(* CODESYS project CtaSysConfig_2.0.0.0.library
   Description: Config Library der CTA
   Version: 2.0.0.0
   Title: CtaSysConfig
   Author: SIS
   DocFormat: reStructuredText
   Placeholder: CtaSysConfig
   LanguageModelAttribute: qualified-access-only
   DefaultNamespace: CtaSysConfig
   CompiledLibraryCompatibilityVersion: CODESYS V3.5 SP16 Patch 3
   Company: CTA

Project tree, tasks and I/O mapping:
  libraries: VisuDialogs, 3.5.16.20 (System); VisuSymbols, 4.5.0.0 (System); SysTypes2 Interfaces, * (System); Util, 3.5.19.0 (System); Standard, 3.5.18.0 (System); StringUtils, 3.5.20.0 (System); SysFile, 3.5.17.0 (System); SysProcess, 3.5.17.0 (System); SysDir, 3.5.17.0 (System); SysTimeRtc, 3.5.20.0 (System); CtaVisSymbols, 2.0.0.0 (CTA); CtaVisUser, 1.0.0.0 (CTA)
  00000000-0000-0000-0000-000000000000|D:\CoDeSys\LibrariesV3\trunk\Intern\CAA\CAA Template\3.5.2.0 draft\Placeholder.xml
  11 Library Parameter/
  30 Program Organization Units/
    08 Bit/
      function block fbSINT [ST]: proValue, proShowValue, metInit, metNewValue, metNewMinMaxNoSave, metNewValueNoSave, proMin, proMax, proStrPara, metNewMinMax, metCheckState
      function block fbBYTE [ST]: proMin, metNewMinMax, proStrPara, metNewValue, proShowValue, metNewValueNoSave, proMax, proValue, metNewMinMaxNoSave, metInit, metCheckState
      function block fbUSINT [ST]: proMax, metNewValueNoSave, proStrPara, metInit, proShowValue, metNewMinMaxNoSave, proValue, proMin, metNewMinMax, metNewValue, metCheckState
    Basis/
      function block fbBackUpConfig [ST]: actCreateDateTime, actCreateFilePath
      function block fbConfigFile [ST]: metLoad, metOpenFile, proErrorNr, metCodeDirCreate, FB_EXIT, metLoadFile, proEventDetekted, metCheckNr, proFilePathCheckFile, metChild, proLoad, metSaveFile, metSave, proError, proFilePath, metCleanUpInit, metInit, FB_INIT, proSave, proInitDone, ProSetInstancePathOnDynCreate, metCleanUp, metCheckLastChild
      function block fbDataType [ST]: proShowValue, proStateChanged, proIsLoading, metInit, proParaNr, proIsSaving, proSaveOnChange, proStrPara, proChildAddDone, metCheckState
    32 Bit/
      function block fbDWORD [ST]: proMin, proStrPara, metNewMinMax, proShowValue, proValue, metInit, metNewMinMaxNoSave, proMax, metNewValue, metNewValueNoSave, metCheckState
      function block fbREAL [ST]: metNewMinMaxNoSave, metNewValueNoSave, proShowValue, proMin, proStrPara, proMax, metInit, metNewValue, proValue, metNewMinMax, metCheckState
      function block fbUDINT [ST]: metNewMinMaxNoSave, proShowValue, metNewValue, metNewValueNoSave, proValue, metNewMinMax, metInit, proMax, proStrPara, proMin, metCheckState
      function block fbTIME [ST]: proValue, proStrPara, proShowValue, metNewValueNoSave, metNewValue, metInit, metNewMinMax, proMin, metNewMinMaxNoSave, proMax, metCheckState
      function block fbDINT [ST]: proStrPara, metInit, metNewValue, proValue, metNewMinMax, proMin, metNewMinMaxNoSave, proMax, proShowValue, metNewValueNoSave, metCheckState
      function block fbTOD [ST]: proStrPara, metInit, metNewMinMax, proMin, proValue, metNewValueNoSave, metNewMinMaxNoSave, metNewValue, proShowValue, proMax, metCheckState
      function block fbDATE_AND_TIME [ST]: metNewMinMax, proMax, proStrPara, proValue, metInit, proShowValue, metNewMinMaxNoSave, proMin, metNewValue, metNewValueNoSave, metCheckState
    64 Bit/
      function block fbLTIME [ST]: proValue, metNewValue, metInit, proMin, metNewValueNoSave, proShowValue, metNewMinMax, proStrPara, proMax, metNewMinMaxNoSave, metCheckState
    1 Bit/
      function block fbBOOL [ST]: proShowValue, metNewValue, proValue, proStrPara, metInit, metNewValueNoSave, proMax, proMin, metCheckState
    16 Bit/
      function block fbINT [ST]: proShowValue, metNewValueNoSave, metInit, proValue, proMin, proStrPara, proMax, metNewValue, metNewMinMax, metNewMinMaxNoSave, metCheckState
      function block fbWORD [ST]: proMax, proStrPara, metNewValue, proMin, metNewMinMax, metInit, proValue, proShowValue, metNewValueNoSave, metNewMinMaxNoSave, metCheckState
      function block fbUINT [ST]: metNewMinMaxNoSave, proMin, metNewValueNoSave, proMax, proStrPara, proValue, metInit, metNewMinMax, metNewValue, proShowValue, metCheckState
    40 Byte String/
      function block fbSTRING40 [ST]: proStrPara, metNewValueNoSave, metInit, proShowValue, proValue, metNewValue, metCheckState
    Functions/
      function fcFileClose [ST]
      function fcGetMin [ST]
      function fcFileOpen [ST]
      function fcGetValueFromDataType [ST]
      function fcRealToString [ST]
      function fcGetValue [ST]
      function fcGetEnumerationId [ST]
      function fcFillStr [ST]
      function fcGetMax [ST]
      function fcFileDelete [ST]
    function FuGetLocalDateAndTime [ST]
  13 Globale Variablen/
    global variables GVL_Config
  00000000-0000-0000-0000-000000000000|D:\CoDeSys\LibrariesV3\trunk\Intern\CAA\CAA Template\3.4.0.0 draft\Placeholder.xml
  12 Konstanten/
    global variables GlobalKonstant
  40 Visualizations/
    32 Bit/
      UDINT/
        visualisation visUDINT
        visualisation visUDINT_QUERRY
        visualisation visUDINT_ITF
      DINT/
        visualisation visDINT_QUERRY
        visualisation visDINT
        visualisation visDINT_ITF
      REAL/
        visualisation visREAL_QUERRY
        visualisation visREAL
        visualisation visREAL_ITF
      TIME/
        visualisation visTIME
        visualisation visTIME_ITF
        visualisation visTIME_QUERRY
      TOD/
        visualisation visTOD_ITF
        visualisation visTOD
        visualisation visTOD_QUERRY
      DWORD/
        DWORD DEZ/
          visualisation visDWORD_QUERRY_DEZ
          visualisation visDWORD_ITF_DEZ
          visualisation visDWORD_DEZ
        DWORD HEX/
          visualisation visDWORD_HEX
          visualisation visDWORD_ITF_HEX
          visualisation visDWORD_QUERRY_HEX
      DATE AND TIME/
        visualisation visDATE_AND_TIME_ITF
        visualisation visDATE_AND_TIME
        visualisation visDATE_AND_TIME_QUERRY
    8 Bit/
      USINT/
        visualisation visUSINT_QUERRY
        visualisation visUSINT_ITF
        visualisation visUSINT
      BYTE/
        visualisation visBYTE_ITF
        visualisation visBYTE
        visualisation visBYTE_QUERRY
      SINT/
        visualisation visSINT_QUERRY
        visualisation visSINT_ITF
        visualisation visSINT
    16 Bit/
      WORD/
        WORD HEX/
          visualisation visWORD_HEX
          visualisation visWORD_QUERRY_HEX
          visualisation visWORD_ITF_HEX
        WORD DEZ/
          visualisation visWORD_ITF_DEZ
          visualisation visWORD_QUERRY_DEZ
          visualisation visWORD_DEZ
      INT/
        visualisation visINT
        visualisation visINT_ITF
        visualisation visINT_QUERRY
      UINT/
        visualisation visUINT
        visualisation visUINT_ITF
        visualisation visUINT_QUERRY
    40 Byte String/
      visualisation visSTRING40_QUERRY
      visualisation visSTRING40
      visualisation visSTRING40_ITF
    ENUMERATION/
      32 Bit/
        visualisation visENUMERATION_DINT_QUERRY
        visualisation visENUMERATION_DINT
      16 Bit/
        visualisation visENUMERATION_INT
        visualisation visENUMERATION_INT_QUERRY
      visualisation visENUMERATION
      8 Bit/
        visualisation visENUMERATION_BYTE
        visualisation visENUMERATION_BYTE_QUERR
    64 Bit/
      LTIME/
        visualisation visLTIME_ITF
        visualisation visLTIME
        visualisation visLTIME_QUERRY
    1 Bit/
      visualisation visBOOL
      visualisation visBOOL_ITF
      visualisation visBOOL_QUERRY
    Show Data/
      visualisation visSHOWDATA_QUERRY
      visualisation visSHOWDATA
      visualisation visSHOWDATA_ITF
  21 Interface/
    16 Bit/
      interface ITF_WORD: proMax, proMin, proValue
      interface ITF_UINT: proMin, proMax, proValue
      interface ITF_INT: proValue, proMin, proMax
    1 Bit/
      interface ITF_BOOL: proValue
    32 Bit/
      interface ITF_REAL: proValue, proMax, proMin
      interface ITF_TIME: proValue, proMax, proMin
      interface ITF_TOD: proValue, proMin, proMax
      interface ITF_DATE_AND_TIME: proMax, proValue, proMin
      interface ITF_UDINT: proMin, proMax, proValue
      interface ITF_DINT: proMax, proMin, proValue
      interface ITF_DWORD: proMin, proValue, proMax
    08 Bit/
      interface ITF_SINT: proValue, proMax, proMin
      interface ITF_BYTE: proMax, proValue, proMin
      interface ITF_USINT: proMin, proValue, proMax
    40 Byte String/
      interface ITF_STRING40: proValue
    Basis/
      interface ITF_DATATYPE: proStrPara, proChildAddDone, proStateChanged, proShowValue, proIsSaving, metInit, proSaveOnChange, proParaNr, proIsLoading
      interface ITF_CONFIGFILE: proLoad, metInit, metSave, proInitDone, metLoad, proSave, metCheckLastChild
    64 Bit/
      interface ITF_LTIME: proValue, proMin, proMax
  60 Textlisten/
  20 Structs/
    data type scStateDataType
    data type scStateConfigFile
  text list GlobalTextList
  50 Images/
  10 Documenation/
    global variables VersionHistory
    global variables readMe
  00000000-0000-0000-0000-000000000000|D:\CoDeSys\LibrariesV3\trunk\Intern\CAA\CAA Template\3.2.0.3 draft\Prefix.pdf
*)

// 20 Structs/scStateDataType
TYPE scStateDataType :
    STRUCT
        xInitDoneDataType       :   BIT;
        xInitDoneConfig         :   BIT;
        xUpdateOldValueNoSave   :   BIT;
        xSaveOnChange           :   BIT; 
        xIsSaving               :   BIT;
        xIsLoading              :   BIT; 
		xStateChanged			:	BIT;  
		xChildAddDone			:	BIT;
    END_STRUCT
END_TYPE

// 20 Structs/scStateConfigFile
TYPE scStateConfigFile :
    STRUCT
        xInit                   :   BIT;
		xInitDone				:	BIT;
		xGetChild				:	BIT;
        xEventSave              :   BIT;
        xEventLoad              :   BIT;
        xEventDetekted          :   BIT;
        xIsOpen                 :   BIT;        
    END_STRUCT
END_TYPE

// 12 Konstanten/GlobalKonstant
{attribute 'qualified_only'}
VAR_GLOBAL CONSTANT
    usiFeldLeng     :   USINT   :=    40;
    diStringSize    :   UINT    :=   129;
    diLineSize      :   UINT    :=   131;    
END_VAR

// 10 Documenation/VersionHistory
(* 

.. image:: ../../Images/CTA_Logo.jpg
   :align: right
   :width: 15% 

**Vorlage**   


============ =========== =========== ============================================
**Date**     **Version** **Author**  **Change**
------------ ----------- ----------- --------------------------------------------
04.03.2021   0.0.0.0     SIS         Vorlage erstellt

============ =========== =========== ============================================


*)
VAR_GLOBAL
    stInfo : STRING:= '0.0.0.0, Vorlage, CTA';
END_VAR

// 10 Documenation/readMe
(*

**ReadMe**
 
|	**Empfehlung**
|
|	Dokumentrieren Sie die Library für eine nachhaltige Entwicklung
|     
| *Beispiel*
| 
| Dies ist die Vorlage Library der CTA. Erstellen Sie ihre Library anhand dieser Vorlage.
*)

VAR_GLOBAL
    xReadMeDone              :   BOOL;
END_VAR

// 13 Globale Variablen/GVL_Config
{attribute 'qualified_only'}
VAR_GLOBAL
    stBackUp            :   STRING[30];
    xSave               :   BOOL;
    xLoad               :   BOOL;
    xError              :   BOOL;
    stPath              :   STRING[255];
END_VAR

// 30 Program Organization Units/32 Bit/fbDWORD
FUNCTION_BLOCK fbDWORD EXTENDS fbDataType IMPLEMENTS ITF_DWORD
VAR_INPUT CONSTANT
    _WertInit      :   DWORD;
    _MinInit       :   DWORD;
    _MaxInit       :   DWORD;       
END_VAR
VAR
    dwValue          :   DWORD;   
    dwMin            :   DWORD;
    dwMax            :   DWORD; 
    {attribute 'hide'}
    dwValueOld       :   DWORD; 
    {attribute 'hide'}
    dwMinOld         :   DWORD;
    {attribute 'hide'}
    dwMaxOld         :   DWORD;
END_VAR

(* Call Supper Objekt *)
IF itfConfigFb <> 0 THEN
    SUPER^();
END_IF;

{attribute 'monitoring':='call'}
PROPERTY proMin : DWORD
SET
dwMin := LIMIT(16#0,proMin,16#FFFFFFFF);
END_SET
GET
proMin := dwMin;
END_GET
END_PROPERTY

{attribute 'hide'}
{attribute 'monitoring':='call'}
PROPERTY proStrPara : STRING(129)
// {attribute 'hide'}
SET
proMax    := TO_DWORD(fcGetMax  ( proStrPara));
proMin    := TO_DWORD(fcGetMin  ( proStrPara));
proValue  := TO_DWORD(fcGetValue( proStrPara));
END_SET
GET
proStrPara :=   CONCAT(                    
                CONCAT( 
                CONCAT(
                CONCAT(                 
                CONCAT(                    
                CONCAT( fcfillStr(CONCAT('P',TO_STRING(SUPER^._usiParaNr)),6)       ,
                        ';'                                                         ),
                        fcfillStr(TO_STRING(dwValue),GlobalKonstant.usiFeldLeng)    ),
                        ';'                                                         ),
                        fcfillStr(TO_STRING(dwMin),GlobalKonstant.usiFeldLeng)      ),
                        ';'                                                         ),
                        fcfillStr(TO_STRING(dwMax),GlobalKonstant.usiFeldLeng)      );
END_GET
END_PROPERTY

METHOD metNewMinMax : BOOL
VAR_INPUT
    newMin      :   DWORD;
    newMax      :   DWORD;
END_VAR
IF newMin <> newMax THEN
    proMin      := newMin;
    proMax      := newMax;
    proValue    := dwValue;    
END_IF;
metNewMinMax := TRUE;
END_METHOD

PROPERTY proShowValue : STRING[40]
GET
proShowValue := TO_STRING(dwValue);
END_GET
END_PROPERTY

{attribute 'monitoring':='call'}
PROPERTY proValue : DWORD
GET
proValue := dwValue;
END_GET
SET
dwValue := LIMIT(proMin,proValue,proMax);
END_SET
END_PROPERTY

{attribute 'hide'}
METHOD metInit : BOOL
IF _MinInit <> _MaxInit THEN
    proMin    := _MinInit;
    proMax    := _MaxInit;
ELSE
    proMin    := 16#F;
    proMax    := 16#FFFFFFFF;
END_IF;
    proValue  := _WertInit;
END_METHOD

METHOD metNewMinMaxNoSave : BOOL
VAR_INPUT
    newMinNoSave      :   DWORD;
    newMaxNoSave      :   DWORD;
END_VAR
IF newMinNoSave <> newMaxNoSave THEN
    proMin      := newMinNoSave;
    proMax      := newMaxNoSave;
    proValue    := dwValue;    
    scState.xUpdateOldValueNoSave := TRUE;
END_IF;
metNewMinMaxNoSave := TRUE;
END_METHOD

{attribute 'monitoring':='call'}
PROPERTY proMax : DWORD
SET
dwMax := LIMIT(16#0,proMax,16#FFFFFFFF);
END_SET
GET
proMax := dwMax;
END_GET
END_PROPERTY

METHOD metNewValue : BOOL
VAR_INPUT
    newValue   :   DWORD;
END_VAR
proValue := newValue;
metNewValue := TRUE;
END_METHOD

METHOD metNewValueNoSave : BOOL
VAR_INPUT
    newValueNoSave   :   DWORD;
END_VAR
proValue := newValueNoSave;
scState.xUpdateOldValueNoSave := TRUE;
metNewValueNoSave := TRUE;
END_METHOD

{attribute 'hide'}
METHOD metCheckState : BOOL
(* Search Change & Save Old Values *)
IF dwValue <> dwValueOld OR dwMin <> dwMinOld OR dwMax <> dwMaxOld OR scState.xUpdateOldValueNoSave THEN
    (* Prüfen ob die Werte bei änderung gespeichert werden sollen *)
    IF scState.xUpdateOldValueNoSave THEN
        scState.xUpdateOldValueNoSave := FALSE;
    ELSE
        proSaveOnChange 	:= TRUE;
	END_IF
	(*State Changed*) 
	scState.xStateChanged 	:= TRUE;   
    proValue   				:= dwValue;
    dwValueOld 				:= proValue;
    proMin     				:= dwMin;
    proMax     				:= dwMax;        
    dwMinOld   				:= proMin;
    dwMaxOld   				:= proMax;
ELSE
	(*State Changed*) 
	scState.xStateChanged 	:= FALSE;    
END_IF;
END_METHOD

END_FUNCTION_BLOCK

// 30 Program Organization Units/Basis/fbDataType
{attribute 'hide_all_locals'}
FUNCTION_BLOCK fbDataType IMPLEMENTS ITF_DATATYPE
VAR_INPUT
    _usiParaNr              :   USINT;
    itfConfigFb             :   ITF_CONFIGFILE;   
END_VAR
VAR
    scState                 :   scStateDataType;
    itfConfigFbSync         :   ITF_CONFIGFILE;
END_VAR

IF itfConfigFb <> 0 THEN
	IF itfConfigFbSync = 0 THEN
		__QUERYINTERFACE(itfConfigFb,itfConfigFbSync);
	END_IF;
	IF itfConfigFb = itfConfigFbSync THEN
		THIS^.metCheckState();
		IF NOT scState.xInitDoneDataType THEN
			THIS^.metInit();
			scState.xInitDoneDataType := TRUE;
		END_IF;
		IF itfConfigFb.proInitDone THEN    
			IF itfConfigFb.proLoad THEN
				itfConfigFb.metLoad(THIS^);
			END_IF;
			IF itfConfigFb.proSave OR scState.xSaveOnChange THEN
				itfConfigFb.metSave(THIS^);
			END_IF;
			itfConfigFb.metCheckLastChild(THIS^);
		ELSIF NOT scState.xInitDoneConfig THEN
			IF itfConfigFb.metInit(THIS^) THEN
				scState.xInitDoneConfig         := TRUE;
				scState.xUpdateOldValueNoSave   := TRUE;
			END_IF;
		END_IF;
	END_IF;    
END_IF;
(* Delete itfConfigFb *)
itfConfigFb := 0;

PROPERTY proShowValue : STRING[40]
GET
proShowValue := '';
END_GET
END_PROPERTY

{attribute 'monitoring':='call'}
PROPERTY proStateChanged : BOOL
GET
proStateChanged := scState.xStateChanged;
END_GET
END_PROPERTY

PROPERTY proIsLoading : BOOL
SET
scState.xIsLoading :=proIsLoading;
END_SET
GET
proIsLoading := scState.xIsLoading;
END_GET
END_PROPERTY

{attribute 'hide'}
METHOD metInit : BOOL
END_METHOD

{attribute 'monitoring':='call'}
PROPERTY proParaNr : USINT
GET
proParaNr := LIMIT(1,_usiParaNr,255);
END_GET
END_PROPERTY

PROPERTY proIsSaving : BOOL
SET
scState.xIsSaving := proIsSaving;
END_SET
GET
proIsSaving := scState.xIsSaving;
END_GET
END_PROPERTY

{attribute 'hide'}
{attribute 'monitoring':='call'}
PROPERTY proSaveOnChange : BOOL
SET
scState.xSaveOnChange := proSaveOnChange;
END_SET
GET
proSaveOnChange := scState.xSaveOnChange;
END_GET
END_PROPERTY

{attribute 'hide'}
{attribute 'monitoring':='call'}
PROPERTY proStrPara : STRING[129]
SET
END_SET
GET
END_GET
END_PROPERTY

PROPERTY proChildAddDone : BOOL
SET
scState.xChildAddDone := proChildAddDone;
END_SET
GET
proChildAddDone := scState.xChildAddDone;
END_GET
END_PROPERTY

{attribute 'hide'}
METHOD metCheckState : BOOL
END_METHOD

END_FUNCTION_BLOCK

// 21 Interface/Basis/ITF_DATATYPE
INTERFACE ITF_DATATYPE EXTENDS __SYSTEM.IQueryInterface

{attribute 'hide'}
{attribute 'monitoring':='call'}
PROPERTY proStrPara : STRING[129]
// {attribute 'hide'}
(*
(* Get *)
(* Tabellenaufbau
+-----+------+------+------+
| PNr | Wert | Min  | Max  |
+-----+------+------+------+
| 6By ; 40By ; 40By ; 40By | = 129By
+-----+------+------+------+
*)
proStrPara :=   CONCAT(                    
                CONCAT( 
                CONCAT(
                CONCAT(                 
                CONCAT(                    
                CONCAT( fcfillStr(CONCAT('P',TO_STRING(_usiParaNr)),5)  ,
                        ';'                                                 ),
                        fcfillStr(TO_STRING(rValue),Konstant.usiFeldLeng)   ),
                        ';'                                                 ),
                        fcfillStr(TO_STRING(rMin),Konstant.usiFeldLeng)     ),
                        ';'                                                 ),
                        fcfillStr(TO_STRING(rMax),Konstant.usiFeldLeng)     );    
                        
                        
                        
(* Set *)
rValue  := TO_REAL(MID(proStrPara,Konstant.usiFeldLeng,7 + (Konstant.usiFeldLeng * 1)+ 0));
rMin    := TO_REAL(MID(proStrPara,Konstant.usiFeldLeng,7 + (Konstant.usiFeldLeng * 2)+ 1));
rMax    := TO_REAL(MID(proStrPara,Konstant.usiFeldLeng,7 + (Konstant.usiFeldLeng * 3)+ 2));                      
                                                
*)
SET
END_SET
GET
END_GET
END_PROPERTY

PROPERTY proChildAddDone : BOOL
GET
END_GET
SET
END_SET
END_PROPERTY

{attribute 'monitoring':='call'}
PROPERTY proStateChanged : BOOL
GET
END_GET
END_PROPERTY

PROPERTY proShowValue : STRING[40]
GET
END_GET
END_PROPERTY

PROPERTY proIsSaving : BOOL
GET
END_GET
SET
END_SET
END_PROPERTY

{attribute 'hide'}
METHOD metInit : BOOL
VAR_INPUT
END_VAR
END_METHOD

{attribute 'monitoring':='call'}
PROPERTY proSaveOnChange : BOOL
SET
END_SET
GET
END_GET
END_PROPERTY

{attribute 'hide'}
{attribute 'monitoring':='call'}
PROPERTY proParaNr : USINT
GET
END_GET
END_PROPERTY

PROPERTY proIsLoading : BOOL
GET
END_GET
SET
END_SET
END_PROPERTY

END_INTERFACE

// 30 Program Organization Units/Functions/fcFillStr
FUNCTION fcFillStr : STRING[GlobalKonstant.usiFeldLeng]
VAR_INPUT
	{attribute 'monitoring_encoding' := 'UTF-8'}
    stIn           : STRING[GlobalKonstant.usiFeldLeng];
    uiLen          : UINT;
END_VAR
VAR
    ui : UINT;
END_VAR

fcFillStr := '';
fcFillStr := stIn;
IF TO_UINT(LEN(stIn)) < uiLen THEN
    FOR ui := LIMIT(0,TO_UINT(LEN(stIn)),LIMIT(0,uiLen,GlobalKonstant.usiFeldLeng)) TO LIMIT(0,uiLen-1,GlobalKonstant.usiFeldLeng) DO
        IF ui = TO_UINT(LEN(stIn)) THEN
            fcFillStr[ui]       := 124; // Trennzeichen
        ELSE
            fcFillStr[ui]       := 32;  // Lehrzeichen
        END_IF; 
        fcFillStr[ui+1]     := 0;  // ClearByte
    END_FOR;
END_IF;

END_FUNCTION

// 21 Interface/Basis/ITF_CONFIGFILE
INTERFACE ITF_CONFIGFILE EXTENDS __SYSTEM.IQueryInterface

{attribute 'monitoring':='call'}
PROPERTY proLoad : BOOL
GET
END_GET
END_PROPERTY

METHOD metInit : BOOL
VAR_INPUT
    itfDataTypeObj  :   ITF_DATATYPE;
END_VAR
END_METHOD

METHOD metSave : BOOL
VAR_INPUT
    itfDataTypeObj  :   ITF_DATATYPE;
END_VAR
END_METHOD

{attribute 'monitoring':='call'}
PROPERTY proInitDone : BOOL
GET
END_GET
END_PROPERTY

METHOD metLoad : BOOL
VAR_INPUT
    itfDataTypeObj  :   ITF_DATATYPE;
END_VAR
END_METHOD

{attribute 'monitoring':='call'}
PROPERTY proSave : BOOL
GET
END_GET
END_PROPERTY

METHOD metCheckLastChild
VAR_INPUT  
    itfDataTypeObj  :   ITF_DATATYPE;
END_VAR
END_METHOD

END_INTERFACE

// 21 Interface/32 Bit/ITF_DWORD
INTERFACE ITF_DWORD EXTENDS ITF_DATATYPE

{attribute 'monitoring':='call'}
PROPERTY proMin : DWORD
SET
END_SET
GET
END_GET
END_PROPERTY

{attribute 'monitoring':='call'}
PROPERTY proValue : DWORD
SET
END_SET
GET
END_GET
END_PROPERTY

{attribute 'monitoring':='call'}
PROPERTY proMax : DWORD
GET
END_GET
SET
END_SET
END_PROPERTY

END_INTERFACE

// 30 Program Organization Units/Functions/fcGetMax
FUNCTION fcGetMax : STRING[40]
VAR_INPUT
	{attribute 'monitoring_encoding' := 'UTF-8'}
    stStrPara   :   STRING[170];    
END_VAR
VAR
END_VAR

fcGetMax                    := (MID(stStrPara,GlobalKonstant.usiFeldLeng,7 + (GlobalKonstant.usiFeldLeng * 2)+ 3));
(* Abschlusszeichen Finden *)
IF FIND(fcGetMax,'|') <> 0 THEN
    fcGetMax                := LEFT(fcGetMax,FIND(fcGetMax,'|')-1);
END_IF;
fcGetMax[LEN(fcGetMax)]     := 0;

END_FUNCTION

// 30 Program Organization Units/Functions/fcGetMin
FUNCTION fcGetMin : STRING[40]
VAR_INPUT
	{attribute 'monitoring_encoding' := 'UTF-8'}
    stStrPara   :   STRING[170];    
END_VAR
VAR
END_VAR

fcGetMin                    := (MID(stStrPara,GlobalKonstant.usiFeldLeng,7 + (GlobalKonstant.usiFeldLeng * 1)+ 2));
(* Abschlusszeichen Finden *)
IF FIND(fcGetMin,'|') <> 0 THEN
    fcGetMin                := LEFT(fcGetMin,FIND(fcGetMin,'|')-1);
END_IF;
fcGetMin[LEN(fcGetMin)]     := 0;

END_FUNCTION

// 30 Program Organization Units/Functions/fcGetValue
{attribute 'hide'}
FUNCTION fcGetValue : STRING[GlobalKonstant.usiFeldLeng]
VAR_INPUT
	{attribute 'monitoring_encoding' := 'UTF-8'}
    stStrPara   :   STRING[126];
END_VAR
VAR
END_VAR

fcGetValue                      := MID(stStrPara,GlobalKonstant.usiFeldLeng,7 + 1);
(* Abschlusszeichen Finden *)
IF FIND(fcGetValue,'|') <> 0 THEN
    fcGetValue                  := LEFT(fcGetValue,FIND(fcGetValue,'|')-1);   
END_IF;
fcGetValue[LEN(fcGetValue)]     := 0;

END_FUNCTION

// 30 Program Organization Units/08 Bit/fbSINT
FUNCTION_BLOCK fbSINT EXTENDS fbDataType IMPLEMENTS ITF_SINT
VAR_INPUT CONSTANT
    _WertInit      :   SINT;
    _MinInit       :   SINT;
    _MaxInit       :   SINT;       
END_VAR
VAR
    siValue          :   SINT;   
    siMin            :   SINT;
    siMax            :   SINT; 
    {attribute 'hide'}
    siValueOld       :   SINT;
    {attribute 'hide'}
    siMinOld         :   SINT;
    {attribute 'hide'}
    siMaxOld         :   SINT; 
END_VAR

(* Call Supper Objekt *)
IF itfConfigFb <> 0 THEN
    SUPER^();
END_IF;

{attribute 'monitoring':='call'}
PROPERTY proValue : sINT
SET
siValue := LIMIT(proMin,proValue,proMax);
END_SET
GET
proValue := siValue;
END_GET
END_PROPERTY

PROPERTY proShowValue : STRING[40]
GET
proShowValue := TO_STRING(siValue);
END_GET
END_PROPERTY

{attribute 'hide'}
METHOD metInit : BOOL
IF _MinInit <> _MaxInit THEN
    proMin    := _MinInit;
    proMax    := _MaxInit;
ELSE
    proMin    :=  -128;
    proMax    :=   127;
END_IF;
    proValue  := _WertInit;
END_METHOD

METHOD metNewValue : BOOL
VAR_INPUT
    newValue   :   SINT;
END_VAR
proValue := newValue;
metNewValue := TRUE;
END_METHOD

METHOD metNewMinMaxNoSave : BOOL
VAR_INPUT
    newMinNoSave      :   SINT;
    newMaxNoSave      :   SINT;
END_VAR
IF newMinNoSave <> newMaxNoSave THEN
    proMin      := newMinNoSave;
    proMax      := newMaxNoSave;
    proValue    := siValue;    
    scState.xUpdateOldValueNoSave := TRUE;
END_IF;
metNewMinMaxNoSave := TRUE;
END_METHOD

METHOD metNewValueNoSave : BOOL
VAR_INPUT
    newValueNoSave   :   SINT;
END_VAR
proValue := newValueNoSave;
scState.xUpdateOldValueNoSave := TRUE;
metNewValueNoSave := TRUE;
END_METHOD

{attribute 'monitoring':='call'}
PROPERTY proMin : sINT
SET
siMin := LIMIT(-128,proMin,127);
END_SET
GET
proMin := siMin;
END_GET
END_PROPERTY

{attribute 'monitoring':='call'}
PROPERTY proMax : sINT
GET
proMax := siMax;
END_GET
SET
siMax := LIMIT(-128,proMax,127);
END_SET
END_PROPERTY

{attribute 'hide'}
{attribute 'monitoring':='call'}
PROPERTY proStrPara : STRING(129)
// {attribute 'hide'}
SET
proMax    := TO_SINT(fcGetMax  ( proStrPara));
proMin    := TO_SINT(fcGetMin  ( proStrPara));
proValue  := TO_SINT(fcGetValue( proStrPara));
END_SET
GET
proStrPara :=   CONCAT(                    
                CONCAT( 
                CONCAT(
                CONCAT(                 
                CONCAT(                    
                CONCAT( fcfillStr(CONCAT('P',TO_STRING(SUPER^._usiParaNr)),6)    ,
                        ';'                                                     ),
                        fcfillStr(TO_STRING(siValue),GlobalKonstant.usiFeldLeng)),
                        ';'                                                     ),
                        fcfillStr(TO_STRING(siMin),GlobalKonstant.usiFeldLeng)  ),
                        ';'                                                     ),
                        fcfillStr(TO_STRING(siMax),GlobalKonstant.usiFeldLeng)  );
END_GET
END_PROPERTY

METHOD metNewMinMax : BOOL
VAR_INPUT
    newMin      :   SINT;
    newMax      :   SINT;
END_VAR
IF newMin <> newMax THEN
    proMin      := newMin;
    proMax      := newMax;
    proValue    := siValue;    
END_IF;
metNewMinMax := TRUE;
END_METHOD

{attribute 'hide'}
METHOD metCheckState : BOOL
(* Search Change & Save Old Values *)
IF siValue <> siValueOld OR siMin <> siMinOld OR siMax <> siMaxOld OR scState.xUpdateOldValueNoSave THEN
    (* Prüfen ob die Werte bei änderung gespeichert werden sollen *)
    IF scState.xUpdateOldValueNoSave THEN
        scState.xUpdateOldValueNoSave := FALSE;
    ELSE
        proSaveOnChange 	:= TRUE;
	END_IF
	(*State Changed*) 
	scState.xStateChanged 	:= TRUE;   
    proValue  				:= siValue;
    siValueOld 				:= proValue;
    proMin     				:= siMin;
    proMax     				:= siMax;    
    siMinOld   				:= proMin;
    siMaxOld   				:= proMax;
ELSE
	(*State Changed*) 
	scState.xStateChanged 	:= FALSE;    
END_IF;
END_METHOD

END_FUNCTION_BLOCK

// 21 Interface/08 Bit/ITF_SINT
INTERFACE ITF_SINT EXTENDS ITF_DATATYPE

{attribute 'monitoring':='call'}
PROPERTY proValue : sINT
SET
END_SET
GET
END_GET
END_PROPERTY

{attribute 'monitoring':='call'}
PROPERTY proMax : sINT
SET
END_SET
GET
END_GET
END_PROPERTY

{attribute 'monitoring':='call'}
PROPERTY proMin : sINT
GET
END_GET
SET
END_SET
END_PROPERTY

END_INTERFACE

// 30 Program Organization Units/32 Bit/fbREAL
FUNCTION_BLOCK fbREAL EXTENDS fbDataType IMPLEMENTS ITF_REAL
VAR_INPUT CONSTANT
    _WertInit      :   REAL;
    _MinInit       :   REAL;
    _MaxInit       :   REAL;       
END_VAR
VAR
    rValue          :   REAL;   
    rMin            :   REAL;
    rMax            :   REAL; 
    {attribute 'hide'}
    rValueOld       :   REAL; 
    {attribute 'hide'}
    rMinOld         :   REAL;
    {attribute 'hide'}
    rMaxOld         :   REAL;
END_VAR

(* Call Supper Objekt *)
IF itfConfigFb <> 0 THEN
    SUPER^();
END_IF;

METHOD metNewMinMaxNoSave : BOOL
VAR_INPUT
    newMinNoSave      :   REAL;
    newMaxNoSave      :   REAL;
END_VAR
IF newMinNoSave <> newMaxNoSave THEN
    proMin      := newMinNoSave;
    proMax      := newMaxNoSave;
    proValue    := rValue;    
    scState.xUpdateOldValueNoSave := TRUE;
END_IF;
metNewMinMaxNoSave := TRUE;
END_METHOD

METHOD metNewValueNoSave : BOOL
VAR_INPUT
    newValueNoSave   :   REAL;
END_VAR
proValue := newValueNoSave;
scState.xUpdateOldValueNoSave := TRUE;
metNewValueNoSave := TRUE;
END_METHOD

PROPERTY proShowValue : STRING[40]
GET
proShowValue := TO_STRING(rValue);
END_GET
END_PROPERTY

{attribute 'monitoring':='call'}
PROPERTY proMin : REAL
SET
rMin := LIMIT(-3.402823E+38,proMin,3.402823E+38);
END_SET
GET
proMin := rMin;
END_GET
END_PROPERTY

{attribute 'hide'}
{attribute 'monitoring':='call'}
PROPERTY proStrPara : STRING[129]
GET
proStrPara :=   CONCAT(                    
                CONCAT( 
                CONCAT(
                CONCAT(                 
                CONCAT(                    
                CONCAT( fcfillStr(CONCAT('P',TO_STRING(SUPER^._usiParaNr)),6)       ,
                        ';'                                                         ),
                        fcfillStr(TO_STRING(rValue),GlobalKonstant.usiFeldLeng)     ),
                        ';'                                                         ),
                        fcfillStr(TO_STRING(rMin),GlobalKonstant.usiFeldLeng)       ),
                        ';'                                                         ),
                        fcfillStr(TO_STRING(rMax),GlobalKonstant.usiFeldLeng)       );
END_GET
SET
proMax    := TO_REAL(fcGetMax  ( proStrPara));
proMin    := TO_REAL(fcGetMin  ( proStrPara));
proValue  := TO_REAL(fcGetValue( proStrPara));
END_SET
END_PROPERTY

{attribute 'monitoring':='call'}
PROPERTY proMax : REAL
SET
rMax := LIMIT(-3.402823E+38,proMax,3.402823E+38);
END_SET
GET
proMax := rMax;
END_GET
END_PROPERTY

{attribute 'hide'}
METHOD metInit : BOOL
IF _MinInit <> _MaxInit THEN
    proMin    := _MinInit;
    proMax    := _MaxInit;
ELSE
    proMin    := -3.402823E+38;
    proMax    :=  3.402823E+38;
END_IF;
    proValue  := _WertInit;
END_METHOD

METHOD metNewValue : BOOL
VAR_INPUT
    newValue   :   REAL;
END_VAR
proValue := newValue;
metNewValue := TRUE;
END_METHOD

{attribute 'monitoring':='call'}
PROPERTY proValue : REAL
SET
rValue := LIMIT(proMin,proValue,proMax);
END_SET
GET
proValue := LIMIT(rMin,rValue,rMax);
END_GET
END_PROPERTY

METHOD metNewMinMax : BOOL
VAR_INPUT
    newMin      :   REAL;
    newMax      :   REAL;
END_VAR
IF newMin <> newMax THEN
    proMin      := newMin;
    proMax      := newMax;
    proValue    := rValue;    
END_IF;
metNewMinMax := TRUE;
END_METHOD

{attribute 'hide'}
METHOD metCheckState : BOOL
(* Search Change & Save Old Values *)
IF rValue <> rValueOld OR rMin <> rMinOld OR rMax <> rMaxOld OR scState.xUpdateOldValueNoSave THEN
    (* Prüfen ob die Werte bei änderung gespeichert werden sollen *)
    IF scState.xUpdateOldValueNoSave THEN
        scState.xUpdateOldValueNoSave := FALSE;
    ELSE
        proSaveOnChange 	:= TRUE;
	END_IF
	(*State Changed*) 
	scState.xStateChanged 	:= TRUE;   
    proValue  				:= rValue;
    rValueOld 				:= proValue;
    proMin    				:= rMin;
    proMax    				:= rMax;      
    rMinOld   				:= proMin;
    rMaxOld   				:= proMax;
ELSE
	(*State Changed*) 
	scState.xStateChanged 	:= FALSE;      
END_IF;
END_METHOD

END_FUNCTION_BLOCK

// 21 Interface/32 Bit/ITF_REAL
INTERFACE ITF_REAL EXTENDS ITF_DATATYPE

{attribute 'monitoring':='call'}
PROPERTY proValue : REAL
SET
END_SET
GET
END_GET
END_PROPERTY

{attribute 'monitoring':='call'}
PROPERTY proMax : REAL
SET
END_SET
GET
END_GET
END_PROPERTY

{attribute 'monitoring':='call'}
PROPERTY proMin : REAL
SET
END_SET
GET
END_GET
END_PROPERTY

END_INTERFACE

// 30 Program Organization Units/08 Bit/fbBYTE
FUNCTION_BLOCK fbBYTE EXTENDS fbDataType IMPLEMENTS ITF_BYTE
VAR_INPUT CONSTANT
    _WertInit        :   BYTE;
    _MinInit         :   BYTE;
    _MaxInit         :   BYTE;       
END_VAR
VAR
    byValue          :   BYTE;   
    byMin            :   BYTE;
    byMax            :   BYTE; 
    {attribute 'hide'} 
    byValueOld       :   BYTE; 
    {attribute 'hide'} 
    byMinOld         :   BYTE;
    {attribute 'hide'} 
    byMaxOld         :   BYTE; 
END_VAR

(* Call Supper Objekt *)
IF itfConfigFb <> 0 THEN
    SUPER^();
END_IF;

{attribute 'monitoring':='call'}
PROPERTY proMin : BYTE
GET
proMin := byMin;
END_GET
SET
byMin := LIMIT(0,proMin,255);
END_SET
END_PROPERTY

METHOD metNewMinMax : BOOL
VAR_INPUT
    newMin      :   BYTE;
    newMax      :   BYTE;
END_VAR
IF newMin <> newMax THEN
    proMin      := newMin;
    proMax      := newMax;
    proValue    := byValue;    
END_IF;
metNewMinMax := TRUE;
END_METHOD

{attribute 'hide'}
{attribute 'monitoring':='call'}
PROPERTY proStrPara : STRING(129)
// {attribute 'hide'}
GET
proStrPara :=   CONCAT(                    
                CONCAT( 
                CONCAT(
                CONCAT(                 
                CONCAT(                     
                CONCAT( fcfillStr(CONCAT('P',TO_STRING(SUPER^._usiParaNr)),6)    ,
                        ';'                                                     ),
                        fcfillStr(TO_STRING(byValue),GlobalKonstant.usiFeldLeng)),
                        ';'                                                     ),
                        fcfillStr(TO_STRING(byMin),GlobalKonstant.usiFeldLeng)  ),
                        ';'                                                     ),
                        fcfillStr(TO_STRING(byMax),GlobalKonstant.usiFeldLeng)  );
END_GET
SET
proMax    := TO_BYTE(fcGetMax  ( proStrPara));
proMin    := TO_BYTE(fcGetMin  ( proStrPara));
proValue  := TO_BYTE(fcGetValue( proStrPara));
END_SET
END_PROPERTY

METHOD metNewValue : BOOL
VAR_INPUT
    newValue   :   BYTE;
END_VAR
proValue := newValue;
metNewValue := TRUE;
END_METHOD

PROPERTY proShowValue : STRING[40]
GET
proShowValue := TO_STRING(byValue);
END_GET
END_PROPERTY

METHOD metNewValueNoSave : BOOL
VAR_INPUT
    newValueNoSave   :   BYTE;
END_VAR
proValue := newValueNoSave;
scState.xUpdateOldValueNoSave := TRUE;
metNewValueNoSave := TRUE;
END_METHOD

{attribute 'monitoring':='call'}
PROPERTY proMax : BYTE
GET
proMax := byMax;
END_GET
SET
byMax := LIMIT(0,proMax,255);
END_SET
END_PROPERTY

{attribute 'monitoring':='call'}
PROPERTY proValue : BYTE
GET
proValue := byValue;
END_GET
SET
byValue := LIMIT(proMin,proValue,proMax);
END_SET
END_PROPERTY

METHOD metNewMinMaxNoSave : BOOL
VAR_INPUT
    newMinNoSave      :   BYTE;
    newMaxNoSave      :   BYTE;
END_VAR
IF newMinNoSave <> newMaxNoSave THEN
    proMin      := newMinNoSave;
    proMax      := newMaxNoSave;
    proValue    := byValue;    
    scState.xUpdateOldValueNoSave := TRUE;
END_IF;
metNewMinMaxNoSave := TRUE;
END_METHOD

{attribute 'hide'}
METHOD metInit : BOOL
IF _MinInit <> _MaxInit THEN
    proMin    := _MinInit;
    proMax    := _MaxInit;
ELSE
    proMin    :=  0;
    proMax    :=  255;
END_IF;
    proValue  := _WertInit;
END_METHOD

{attribute 'hide'}
METHOD metCheckState : BOOL
(* Search Change & Save Old Values *)
IF byValue <> byValueOld OR byMin <> byMinOld OR byMax <> byMaxOld OR scState.xUpdateOldValueNoSave THEN
    (* Prüfen ob die Werte bei änderung gespeichert werden sollen *)
    IF scState.xUpdateOldValueNoSave THEN
        scState.xUpdateOldValueNoSave := FALSE;
    ELSE
        proSaveOnChange		 := TRUE;
	END_IF
	(*State Changed*) 
	scState.xStateChanged 	:= TRUE;  
    proValue   				:= byValue;
    byValueOld 				:= proValue;
    proMin     				:= byMin;
    proMax     				:= byMax;       
    byMinOld   				:= proMin;
    byMaxOld   				:= proMax;
ELSE
	(*State Changed*) 
	scState.xStateChanged 	:= FALSE;    
END_IF;
END_METHOD

END_FUNCTION_BLOCK

// 21 Interface/08 Bit/ITF_BYTE
INTERFACE ITF_BYTE EXTENDS ITF_DATATYPE

{attribute 'monitoring':='call'}
PROPERTY proMax : BYTE
GET
END_GET
SET
END_SET
END_PROPERTY

{attribute 'monitoring':='call'}
PROPERTY proValue : BYTE
GET
END_GET
SET
END_SET
END_PROPERTY

{attribute 'monitoring':='call'}
PROPERTY proMin : BYTE
SET
END_SET
GET
END_GET
END_PROPERTY

END_INTERFACE

// 21 Interface/1 Bit/ITF_BOOL
INTERFACE ITF_BOOL EXTENDS ITF_DATATYPE

{attribute 'monitoring':='call'}
PROPERTY proValue : BOOL
GET
END_GET
SET
END_SET
END_PROPERTY

END_INTERFACE

// 30 Program Organization Units/Functions/fcFileClose
FUNCTION fcFileClose : RTS_IEC_RESULT
VAR_INPUT
    hFile   :   RTS_IEC_HANDLE;
	stPath	:	STRING(255);
	stMeth	:	STRING(50);
END_VAR
VAR
END_VAR

IF hFile <> 0 THEN
    fcFileClose := SysFile.SysFileClose(hFile);
END_IF;

END_FUNCTION

// 30 Program Organization Units/Functions/fcFileOpen
FUNCTION fcFileOpen : RTS_IEC_HANDLE
VAR_INPUT
	{attribute 'monitoring_encoding' := 'UTF-8'}
    stFilePath  :   STRING[255];
    AccesMode   :   ACCESS_MODE;
    refResult   :   REFERENCE TO RTS_IEC_RESULT;
END_VAR

fcFileOpen := SysFile.SysFileOpen(stFilePath,AccesMode,ADR(refResult));

END_FUNCTION

// 30 Program Organization Units/16 Bit/fbINT
FUNCTION_BLOCK fbINT EXTENDS fbDataType IMPLEMENTS ITF_INT
VAR_INPUT CONSTANT
    _WertInit      :   INT;
    _MinInit       :   INT;
    _MaxInit       :   INT;       
END_VAR
VAR
    iValue          :   INT;   
    iMin            :   INT;
    iMax            :   INT; 
    {attribute 'hide'}
    iValueOld       :   INT;
    {attribute 'hide'}
    iMinOld         :   INT;
    {attribute 'hide'}
    iMaxOld         :   INT;
END_VAR

(* Call Supper Objekt *)
IF itfConfigFb <> 0 THEN
    SUPER^();
END_IF;

PROPERTY proShowValue : STRING[40]
GET
proShowValue := TO_STRING(iValue);
END_GET
END_PROPERTY

METHOD metNewValueNoSave : BOOL
VAR_INPUT
    newValueNoSave   :   INT;
END_VAR
proValue := newValueNoSave;
scState.xUpdateOldValueNoSave := TRUE;
metNewValueNoSave := TRUE;
END_METHOD

{attribute 'hide'}
METHOD metInit : BOOL
IF _MinInit <> _MaxInit THEN
    proMin    := _MinInit;
    proMax    := _MaxInit;
ELSE
    proMin    :=  -32768;
    proMax    :=   32767;
END_IF;
    proValue  := _WertInit;
END_METHOD

{attribute 'monitoring':='call'}
PROPERTY proValue : INT
SET
iValue := LIMIT(proMin,proValue,proMax);
END_SET
GET
proValue := iValue;
END_GET
END_PROPERTY

{attribute 'monitoring':='call'}
PROPERTY proMin : INT
GET
proMin := iMin;
END_GET
SET
iMin := LIMIT(-32768,proMin,32767);
END_SET
END_PROPERTY

{attribute 'hide'}
{attribute 'monitoring':='call'}
PROPERTY proStrPara : STRING(129)
// {attribute 'hide'}
SET
proMax    := TO_INT(fcGetMax  ( proStrPara));
proMin    := TO_INT(fcGetMin  ( proStrPara));
proValue  := TO_INT(fcGetValue( proStrPara));
END_SET
GET
proStrPara :=   CONCAT(                    
                CONCAT( 
                CONCAT(
                CONCAT(                 
                CONCAT(                    
                CONCAT( fcfillStr(CONCAT('P',TO_STRING(SUPER^._usiParaNr)),6)       ,
                        ';'                                                         ),
                        fcfillStr(TO_STRING(iValue),GlobalKonstant.usiFeldLeng)     ),
                        ';'                                                         ),
                        fcfillStr(TO_STRING(iMin),GlobalKonstant.usiFeldLeng)       ),
                        ';'                                                         ),
                        fcfillStr(TO_STRING(iMax),GlobalKonstant.usiFeldLeng)       );
END_GET
END_PROPERTY

{attribute 'monitoring':='call'}
PROPERTY proMax : INT
GET
proMax := iMax;
END_GET
SET
iMax := LIMIT(-32768,proMax,32767);
END_SET
END_PROPERTY

METHOD metNewValue : BOOL
VAR_INPUT
    newValue   :   INT;
END_VAR
proValue := newValue;
metNewValue := TRUE;
END_METHOD

METHOD metNewMinMax : BOOL
VAR_INPUT
    newMin      :   INT;
    newMax      :   INT;
END_VAR
IF newMin <> newMax THEN
    proMin      := newMin;
    proMax      := newMax;
    proValue    := iValue;    
END_IF;
metNewMinMax := TRUE;
END_METHOD

METHOD metNewMinMaxNoSave : BOOL
VAR_INPUT
    newMinNoSave      :   INT;
    newMaxNoSave      :   INT;
END_VAR
IF newMinNoSave <> newMaxNoSave THEN
    proMin      := newMinNoSave;
    proMax      := newMaxNoSave;
    proValue    := iValue;    
    scState.xUpdateOldValueNoSave := TRUE;
END_IF;
metNewMinMaxNoSave := TRUE;
END_METHOD

{attribute 'hide'}
METHOD metCheckState : BOOL
(* Search Change & Save Old Values *)
IF iValue <> iValueOld OR iMin <> iMinOld OR iMax <> iMaxOld OR scState.xUpdateOldValueNoSave THEN
    (* Prüfen ob die Werte bei änderung gespeichert werden sollen *)
    IF scState.xUpdateOldValueNoSave THEN
        scState.xUpdateOldValueNoSave := FALSE;
    ELSE
        proSaveOnChange 	:= TRUE;
	END_IF
	(*State Changed*) 
	scState.xStateChanged 	:= TRUE;   
    proValue        		:= iValue;
    iValueOld       		:= proValue;
    proMin          		:= iMin;
    proMax          		:= iMax;        
    iMinOld         		:= proMin;
    iMaxOld         		:= proMax;
ELSE
	(*State Changed*) 
	scState.xStateChanged 	:= FALSE;    
END_IF;
END_METHOD

END_FUNCTION_BLOCK

// 21 Interface/16 Bit/ITF_INT
INTERFACE ITF_INT EXTENDS ITF_DATATYPE

{attribute 'monitoring':='call'}
PROPERTY proValue : INT
SET
END_SET
GET
END_GET
END_PROPERTY

{attribute 'monitoring':='call'}
PROPERTY proMin : INT
GET
END_GET
SET
END_SET
END_PROPERTY

{attribute 'monitoring':='call'}
PROPERTY proMax : INT
GET
END_GET
SET
END_SET
END_PROPERTY

END_INTERFACE

// 30 Program Organization Units/32 Bit/fbUDINT
FUNCTION_BLOCK fbUDINT EXTENDS fbDataType IMPLEMENTS ITF_UDINT
VAR_INPUT CONSTANT
    _WertInit      :   UDINT;
    _MinInit       :   UDINT;
    _MaxInit       :   UDINT;       
END_VAR
VAR
    udiValue          :   UDINT;   
    udiMin            :   UDINT;
    udiMax            :   UDINT; 
    {attribute 'hide'}
    udiValueOld       :   UDINT;  
    {attribute 'hide'}
    udiMinOld         :   UDINT;
    {attribute 'hide'}
    udiMaxOld         :   UDINT;
END_VAR

(* Call Supper Objekt *)
IF itfConfigFb <> 0 THEN
    SUPER^();
END_IF;

METHOD metNewMinMaxNoSave : BOOL
VAR_INPUT
    newMinNoSave      :   UDINT;
    newMaxNoSave      :   UDINT;
END_VAR
IF newMinNoSave <> newMaxNoSave THEN
    proMin      := newMinNoSave;
    proMax      := newMaxNoSave;
    proValue    := udiValue;    
    scState.xUpdateOldValueNoSave := TRUE;
END_IF;
metNewMinMaxNoSave := TRUE;
END_METHOD

PROPERTY proShowValue : STRING[40]
GET
proShowValue := TO_STRING(udiValue);
END_GET
END_PROPERTY

METHOD metNewValue : BOOL
VAR_INPUT
    newValue   :   UDINT;
END_VAR
proValue := newValue;
metNewValue := TRUE;
END_METHOD

METHOD metNewValueNoSave : BOOL
VAR_INPUT
    newValueNoSave   :   UDINT;
END_VAR
proValue := newValueNoSave;
scState.xUpdateOldValueNoSave := TRUE;
metNewValueNoSave := TRUE;
END_METHOD

{attribute 'monitoring':='call'}
PROPERTY proValue : UdINT
GET
proValue := udiValue;
END_GET
SET
udiValue := LIMIT(proMin,proValue,proMax);
END_SET
END_PROPERTY

METHOD metNewMinMax : BOOL
VAR_INPUT
    newMin      :   UDINT;
    newMax      :   UDINT;
END_VAR
IF newMin <> newMax THEN
    proMin      := newMin;
    proMax      := newMax;
    proValue    := udiValue;    
END_IF;
metNewMinMax := TRUE;
END_METHOD

{attribute 'hide'}
METHOD metInit : BOOL
IF _MinInit <> _MaxInit THEN
    proMin    := _MinInit;
    proMax    := _MaxInit;
ELSE
    proMin    := 0;
    proMax    := 4294967295;
END_IF;
    proValue  := _WertInit;
END_METHOD

{attribute 'monitoring':='call'}
PROPERTY proMax : UdINT
SET
udiMax := LIMIT(0,proMax,4294967295);
END_SET
GET
proMax := udiMax;
END_GET
END_PROPERTY

{attribute 'hide'}
{attribute 'monitoring':='call'}
PROPERTY proStrPara : STRING(129)
// {attribute 'hide'}
GET
proStrPara :=   CONCAT(                    
                CONCAT( 
                CONCAT(
                CONCAT(                 
                CONCAT(                  
                CONCAT( fcfillStr(CONCAT('P',TO_STRING(SUPER^._usiParaNr)),6)       ,
                        ';'                                                         ),
                        fcfillStr(TO_STRING(udiValue),GlobalKonstant.usiFeldLeng)   ),
                        ';'                                                         ),
                        fcfillStr(TO_STRING(udiMin),GlobalKonstant.usiFeldLeng)     ),
                        ';'                                                         ),
                        fcfillStr(TO_STRING(udiMax),GlobalKonstant.usiFeldLeng)     );
END_GET
SET
proMax    := TO_UDINT(fcGetMax  ( proStrPara));
proMin    := TO_UDINT(fcGetMin  ( proStrPara));
proValue  := TO_UDINT(fcGetValue( proStrPara));
END_SET
END_PROPERTY

{attribute 'monitoring':='call'}
PROPERTY proMin : UdINT
SET
udiMin := LIMIT(0,proMin,4294967295);
END_SET
GET
proMin := udiMin;
END_GET
END_PROPERTY

{attribute 'hide'}
METHOD metCheckState : BOOL
(* Search Change & Save Old Values *)
IF udiValue <> udiValueOld OR udiMin <> udiMinOld OR udiMax <> udiMaxOld OR scState.xUpdateOldValueNoSave THEN
    (* Prüfen ob die Werte bei änderung gespeichert werden sollen *)
    IF scState.xUpdateOldValueNoSave THEN
        scState.xUpdateOldValueNoSave := FALSE;
    ELSE
        proSaveOnChange 	:= TRUE;
	END_IF
	(*State Changed*) 
	scState.xStateChanged 	:= TRUE;   
    proValue        		:= udiValue;
    udiValueOld     		:= proValue;
    proMin          		:= udiMin;
    proMax          		:= udiMax;        
    udiMinOld       		:= proMin;
    udiMaxOld       		:= proMax; 
ELSE
	(*State Changed*) 
	scState.xStateChanged 	:= FALSE;   
END_IF;
END_METHOD

END_FUNCTION_BLOCK

// 21 Interface/32 Bit/ITF_UDINT
INTERFACE ITF_UDINT EXTENDS ITF_DATATYPE

{attribute 'monitoring':='call'}
PROPERTY proMin : UdINT
SET
END_SET
GET
END_GET
END_PROPERTY

{attribute 'monitoring':='call'}
PROPERTY proMax : UdINT
GET
END_GET
SET
END_SET
END_PROPERTY

{attribute 'monitoring':='call'}
PROPERTY proValue : UdINT
SET
END_SET
GET
END_GET
END_PROPERTY

END_INTERFACE

// 21 Interface/32 Bit/ITF_TIME
INTERFACE ITF_TIME EXTENDS ITF_DATATYPE

{attribute 'monitoring':='call'}
PROPERTY proValue : TIME
SET
END_SET
GET
END_GET
END_PROPERTY

{attribute 'monitoring':='call'}
PROPERTY proMax : TIME
GET
END_GET
SET
END_SET
END_PROPERTY

{attribute 'monitoring':='call'}
PROPERTY proMin : TIME
GET
END_GET
SET
END_SET
END_PROPERTY

END_INTERFACE

// 30 Program Organization Units/16 Bit/fbWORD
FUNCTION_BLOCK fbWORD EXTENDS fbDataType IMPLEMENTS ITF_WORD
VAR_INPUT CONSTANT
    _WertInit      :   WORD;
    _MinInit       :   WORD;
    _MaxInit       :   WORD;       
END_VAR
VAR
    wValue          :   WORD;   
    wMin            :   WORD;
    wMax            :   WORD; 
    {attribute 'hide'}
    wValueOld       :   WORD;
    {attribute 'hide'}
    wMinOld         :   WORD;
    {attribute 'hide'}
    wMaxOld         :   WORD;
END_VAR

(* Call Supper Objekt *)
IF itfConfigFb <> 0 THEN
    SUPER^();
END_IF;

{attribute 'monitoring':='call'}
PROPERTY proMax : WORD
GET
proMax := wMax;
END_GET
SET
wMax := LIMIT(16#0,proMax,16#FFFF);
END_SET
END_PROPERTY

{attribute 'hide'}
{attribute 'monitoring':='call'}
PROPERTY proStrPara : STRING(129)
// {attribute 'hide'}
GET
proStrPara :=   CONCAT(                    
                CONCAT( 
                CONCAT(
                CONCAT(                 
                CONCAT(                 
                CONCAT( fcfillStr(CONCAT('P',TO_STRING(SUPER^._usiParaNr)),6)    ,
                        ';'                                                     ),
                        fcfillStr(TO_STRING(wValue),GlobalKonstant.usiFeldLeng) ),
                        ';'                                                     ),
                        fcfillStr(TO_STRING(wMin),GlobalKonstant.usiFeldLeng)   ),
                        ';'                                                     ),
                        fcfillStr(TO_STRING(wMax),GlobalKonstant.usiFeldLeng)   );
END_GET
SET
proMax    := TO_WORD(fcGetMax  ( proStrPara));
proMin    := TO_WORD(fcGetMin  ( proStrPara));
proValue  := TO_WORD(fcGetValue( proStrPara));
END_SET
END_PROPERTY

METHOD metNewValue : BOOL
VAR_INPUT
    newValue   :   WORD;
END_VAR
proValue := newValue;
metNewValue := TRUE;
END_METHOD

{attribute 'monitoring':='call'}
PROPERTY proMin : WORD
GET
proMin := wMin;
END_GET
SET
wMin := LIMIT(16#0,proMin,16#FFFF);
END_SET
END_PROPERTY

METHOD metNewMinMax : BOOL
VAR_INPUT
    newMin      :   WORD;
    newMax      :   WORD;
END_VAR
IF newMin <> newMax THEN
    proMin      := newMin;
    proMax      := newMax;
    proValue    := wValue;    
END_IF;
metNewMinMax := TRUE;
END_METHOD

{attribute 'hide'}
METHOD metInit : BOOL
IF _MinInit <> _MaxInit THEN
    proMin    := _MinInit;
    proMax    := _MaxInit;
ELSE
    proMin    :=  16#0;
    proMax    :=  16#FFFF;
END_IF;
    proValue  := _WertInit;
END_METHOD

{attribute 'monitoring':='call'}
PROPERTY proValue : WORD
SET
wValue := LIMIT(proMin,proValue,proMax);
END_SET
GET
proValue := wValue;
END_GET
END_PROPERTY

PROPERTY proShowValue : STRING[40]
GET
proShowValue := TO_STRING(wValue);
END_GET
END_PROPERTY

METHOD metNewValueNoSave : BOOL
VAR_INPUT
    newValueNoSave   :   WORD;
END_VAR
proValue := newValueNoSave;
scState.xUpdateOldValueNoSave := TRUE;
metNewValueNoSave := TRUE;
END_METHOD

METHOD metNewMinMaxNoSave : BOOL
VAR_INPUT
    newMinNoSave      :   WORD;
    newMaxNoSave      :   WORD;
END_VAR
IF newMinNoSave <> newMaxNoSave THEN
    proMin      := newMinNoSave;
    proMax      := newMaxNoSave;
    proValue    := wValue;    
    scState.xUpdateOldValueNoSave := TRUE;
END_IF;
metNewMinMaxNoSave := TRUE;
END_METHOD

{attribute 'hide'}
METHOD metCheckState : BOOL
(* Search Change & Save Old Values *)
IF wValue <> wValueOld OR wMin <> wMinOld OR wMax <> wMaxOld OR scState.xUpdateOldValueNoSave THEN
    (* Prüfen ob die Werte bei änderung gespeichert werden sollen *)
    IF scState.xUpdateOldValueNoSave THEN
        scState.xUpdateOldValueNoSave := FALSE;
    ELSE
        proSaveOnChange 	:= TRUE;
	END_IF
	(*State Changed*) 
	scState.xStateChanged 	:= TRUE;   
    proValue  				:= wValue;
    wValueOld 				:= proValue;
    proMin    				:= wMin;
    proMax    				:= wMax;
    wMinOld   				:= proMin;
    wMaxOld   				:= proMax;
ELSE
	(*State Changed*) 
	scState.xStateChanged 	:= FALSE;
END_IF;
END_METHOD

END_FUNCTION_BLOCK

// 21 Interface/16 Bit/ITF_WORD
INTERFACE ITF_WORD EXTENDS ITF_DATATYPE

{attribute 'monitoring':='call'}
PROPERTY proMax : WORD
GET
END_GET
SET
END_SET
END_PROPERTY

{attribute 'monitoring':='call'}
PROPERTY proMin : WORD
SET
END_SET
GET
END_GET
END_PROPERTY

{attribute 'monitoring':='call'}
PROPERTY proValue : WORD
SET
END_SET
GET
END_GET
END_PROPERTY

END_INTERFACE

// 21 Interface/32 Bit/ITF_TOD
INTERFACE ITF_TOD EXTENDS ITF_DATATYPE

{attribute 'monitoring':='call'}
PROPERTY proValue : TOD
GET
END_GET
SET
END_SET
END_PROPERTY

{attribute 'monitoring':='call'}
PROPERTY proMin : TOD
GET
END_GET
SET
END_SET
END_PROPERTY

{attribute 'monitoring':='call'}
PROPERTY proMax : TOD
GET
END_GET
SET
END_SET
END_PROPERTY

END_INTERFACE

// 30 Program Organization Units/16 Bit/fbUINT
FUNCTION_BLOCK fbUINT EXTENDS fbDataType IMPLEMENTS ITF_UINT
VAR_INPUT CONSTANT
    _WertInit      :   UINT;
    _MinInit       :   UINT;
    _MaxInit       :   UINT;       
END_VAR
VAR
    uiValue          :   UINT;   
    uiMin            :   UINT;
    uiMax            :   UINT; 
    {attribute 'hide'}
    uiValueOld       :   UINT; 
    {attribute 'hide'}
    uiMinOld         :   UINT;
    {attribute 'hide'}
    uiMaxOld         :   UINT;
END_VAR

(* Call Supper Objekt *)
IF itfConfigFb <> 0 THEN
    SUPER^();
END_IF;

METHOD metNewMinMaxNoSave : BOOL
VAR_INPUT
    newMinNoSave      :   UINT;
    newMaxNoSave      :   UINT;
END_VAR
IF newMinNoSave <> newMaxNoSave THEN
    proMin      := newMinNoSave;
    proMax      := newMaxNoSave;
    proValue    := uiValue;    
    scState.xUpdateOldValueNoSave := TRUE;
END_IF;
metNewMinMaxNoSave := TRUE;
END_METHOD

{attribute 'monitoring':='call'}
PROPERTY proMin : UINT
SET
uiMin := LIMIT(0,proMin,65535);
END_SET
GET
proMin := uiMin;
END_GET
END_PROPERTY

METHOD metNewValueNoSave : BOOL
VAR_INPUT
    newValueNoSave   :   UINT;
END_VAR
proValue := newValueNoSave;
scState.xUpdateOldValueNoSave := TRUE;
metNewValueNoSave := TRUE;
END_METHOD

{attribute 'monitoring':='call'}
PROPERTY proMax : UINT
SET
uiMax := LIMIT(0,proMax,65535);
END_SET
GET
proMax := uiMax;
END_GET
END_PROPERTY

{attribute 'hide'}
{attribute 'monitoring':='call'}
PROPERTY proStrPara : STRING(129)
// {attribute 'hide'}
SET
proMax    := TO_UINT(fcGetMax  ( proStrPara));
proMin    := TO_UINT(fcGetMin  ( proStrPara));
proValue  := TO_UINT(fcGetValue( proStrPara));
END_SET
GET
proStrPara :=   CONCAT(                    
                CONCAT( 
                CONCAT(
                CONCAT(                 
                CONCAT(                  
                CONCAT( fcfillStr(CONCAT('P',TO_STRING(SUPER^._usiParaNr)),6)       ,
                        ';'                                                         ),
                        fcfillStr(TO_STRING(uiValue),GlobalKonstant.usiFeldLeng)    ),
                        ';'                                                         ),
                        fcfillStr(TO_STRING(uiMin),GlobalKonstant.usiFeldLeng)      ),
                        ';'                                                         ),
                        fcfillStr(TO_STRING(uiMax),GlobalKonstant.usiFeldLeng)      );
END_GET
END_PROPERTY

{attribute 'monitoring':='call'}
PROPERTY proValue : UINT
GET
proValue := uiValue;
END_GET
SET
uiValue := LIMIT(proMin,proValue,proMax);
END_SET
END_PROPERTY

{attribute 'hide'}
METHOD metInit : BOOL
IF _MinInit <> _MaxInit THEN
    proMin    := _MinInit;
    proMax    := _MaxInit;
ELSE
    proMin    :=  0;
    proMax    :=  65535;
END_IF;
    proValue  := _WertInit;
END_METHOD

METHOD metNewMinMax : BOOL
VAR_INPUT
    newMin      :   UINT;
    newMax      :   UINT;
END_VAR
IF newMin <> newMax THEN
    proMin      := newMin;
    proMax      := newMax;
    proValue    := uiValue;    
END_IF;
metNewMinMax := TRUE;
END_METHOD

METHOD metNewValue : BOOL
VAR_INPUT
    newValue   :   UINT;
END_VAR
proValue := newValue;
metNewValue := TRUE;
END_METHOD

PROPERTY proShowValue : STRING[40]
GET
proShowValue := TO_STRING(uiValue);
END_GET
END_PROPERTY

{attribute 'hide'}
METHOD metCheckState : BOOL
(* Search Change & Save Old Values *)
IF uiValue <> uiValueOld OR uiMin <> uiMinOld OR uiMax <> uiMaxOld OR scState.xUpdateOldValueNoSave THEN
    (* Prüfen ob die Werte bei änderung gespeichert werden sollen *)
    IF scState.xUpdateOldValueNoSave THEN
        scState.xUpdateOldValueNoSave := FALSE;
    ELSE
        proSaveOnChange		:= TRUE;
	END_IF
	(*State Changed*) 
	scState.xStateChanged 	:= TRUE;   
    proValue   				:= uiValue;
    uiValueOld 				:= proValue;
    proMin     				:= uiMin;
    proMax     				:= uiMax;
    uiMinOld   				:= proMin;
    uiMaxOld   				:= proMax;
ELSE
	(*State Changed*) 
	scState.xStateChanged 	:= FALSE;
END_IF;
END_METHOD

END_FUNCTION_BLOCK

// 21 Interface/16 Bit/ITF_UINT
INTERFACE ITF_UINT EXTENDS ITF_DATATYPE

{attribute 'monitoring':='call'}
PROPERTY proMin : UINT
SET
END_SET
GET
END_GET
END_PROPERTY

{attribute 'monitoring':='call'}
PROPERTY proMax : UINT
GET
END_GET
SET
END_SET
END_PROPERTY

{attribute 'monitoring':='call'}
PROPERTY proValue : UINT
GET
END_GET
SET
END_SET
END_PROPERTY

END_INTERFACE

// 30 Program Organization Units/1 Bit/fbBOOL
FUNCTION_BLOCK fbBOOL EXTENDS fbDataType IMPLEMENTS ITF_BOOL
VAR_INPUT CONSTANT
    _WertInit        :   BOOL;
END_VAR
VAR
    xValue           :   BOOL;   
    {attribute 'hide'} 
    xValueOld        :   BOOL;
END_VAR

(* Call Supper Objekt *)
IF itfConfigFb <> 0 THEN
    SUPER^();
END_IF;

PROPERTY proShowValue : STRING[40]
GET
proShowValue := TO_STRING(xValue);
END_GET
END_PROPERTY

METHOD metNewValue : BOOL
VAR_INPUT
    newValue   :   BOOL;
END_VAR
proValue := newValue;
metNewValue := TRUE;
END_METHOD

{attribute 'monitoring':='call'}
PROPERTY proValue : BOOL
GET
proValue := xValue;
END_GET
SET
xValue := LIMIT(FALSE,proValue,TRUE);
END_SET
END_PROPERTY

{attribute 'hide'}
{attribute 'monitoring':='call'}
PROPERTY proStrPara : STRING(129)
// {attribute 'hide'}
SET
proMax    := TO_BOOL(fcGetMax  ( proStrPara));
proMin    := TO_BOOL(fcGetMin  ( proStrPara));
proValue  := TO_BOOL(fcGetValue( proStrPara));
END_SET
GET
proStrPara :=   CONCAT(                    
                CONCAT( 
                CONCAT(
                CONCAT(                 
                CONCAT(                   
                CONCAT( fcfillStr(CONCAT('P',TO_STRING(SUPER^._usiParaNr)),6)    ,
                        ';'                                                     ),
                        fcfillStr(TO_STRING(xValue),GlobalKonstant.usiFeldLeng) ),
                        ';'                                                     ),
                        fcfillStr(TO_STRING(FALSE),GlobalKonstant.usiFeldLeng)  ),
                        ';'                                                     ),
                        fcfillStr(TO_STRING(TRUE),GlobalKonstant.usiFeldLeng)   );
END_GET
END_PROPERTY

{attribute 'hide'}
METHOD metInit : BOOL
proValue  := _WertInit;
END_METHOD

METHOD metNewValueNoSave : BOOL
VAR_INPUT
    newValueNoSave   :   BOOL;
END_VAR
proValue := newValueNoSave;
scState.xUpdateOldValueNoSave := TRUE;
metNewValueNoSave := TRUE;
END_METHOD

{attribute 'monitoring':='call'}
PROPERTY proMax : BOOL
SET
RETURN;
END_SET
GET
proMax := TRUE;
END_GET
END_PROPERTY

{attribute 'monitoring':='call'}
PROPERTY proMin : BOOL
SET
RETURN;
END_SET
GET
proMin := FALSE;
END_GET
END_PROPERTY

{attribute 'hide'}
METHOD metCheckState : BOOL
(* Search Change & Save Old Values *)
IF xValue <> xValueOld OR scState.xUpdateOldValueNoSave THEN
    (* Prüfen ob die Werte bei änderung gespeichert werden sollen *)
    IF scState.xUpdateOldValueNoSave THEN
        scState.xUpdateOldValueNoSave := FALSE;
    ELSE
        proSaveOnChange 	:= TRUE;
	END_IF
	(*State Changed*) 
	scState.xStateChanged 	:= TRUE;            
    proValue  				:= xValue;
    xValueOld 				:= proValue;
ELSE
	(*State Changed*) 
	scState.xStateChanged 	:= FALSE;
END_IF;
END_METHOD

END_FUNCTION_BLOCK

// 30 Program Organization Units/Functions/fcGetValueFromDataType
FUNCTION fcGetValueFromDataType : STRING[40]
VAR_INPUT
    fbDATATYPEIn     :   ITF_DATATYPE;	
END_VAR
VAR
    fbDATATYPE       :   ITF_DATATYPE;	
END_VAR

IF __QUERYINTERFACE(fbDATATYPEIn,fbDATATYPE) THEN
    fcGetValueFromDataType := fbDATATYPE.proShowValue;
ELSE
    fcGetValueFromDataType := '';
END_IF;

END_FUNCTION

// 21 Interface/32 Bit/ITF_DATE_AND_TIME
INTERFACE ITF_DATE_AND_TIME EXTENDS ITF_DATATYPE

{attribute 'monitoring':='call'}
PROPERTY proMax : DT
GET
END_GET
SET
END_SET
END_PROPERTY

{attribute 'monitoring':='call'}
PROPERTY proValue : DT
GET
END_GET
SET
END_SET
END_PROPERTY

{attribute 'monitoring':='call'}
PROPERTY proMin : DT
GET
END_GET
SET
END_SET
END_PROPERTY

END_INTERFACE

// 30 Program Organization Units/32 Bit/fbTIME
FUNCTION_BLOCK fbTIME EXTENDS fbDataType IMPLEMENTS ITF_TIME
VAR_INPUT CONSTANT
    _WertInit      :   TIME;
    _MinInit       :   TIME;
    _MaxInit       :   TIME;       
END_VAR
VAR
    tValue          :   TIME;   
    tMin            :   TIME;
    tMax            :   TIME; 
    {attribute 'hide'}
    tValueOld       :   TIME;
    {attribute 'hide'}
    tMinOld         :   TIME;
    {attribute 'hide'}
    tMaxOld         :   TIME;
END_VAR

(* Call Supper Objekt *)
IF itfConfigFb <> 0 THEN
    SUPER^();
END_IF;

{attribute 'monitoring':='call'}
PROPERTY proValue : TIME
GET
proValue := LIMIT(tMin,tValue,tMax);
END_GET
SET
tValue := LIMIT(proMin,proValue,proMax);
END_SET
END_PROPERTY

{attribute 'hide'}
{attribute 'monitoring':='call'}
PROPERTY proStrPara : STRING[129]
GET
proStrPara :=   CONCAT(                    
                CONCAT( 
                CONCAT(
                CONCAT(                 
                CONCAT(                  
                CONCAT( fcfillStr(CONCAT('P',TO_STRING(SUPER^._usiParaNr)),6)    ,
                        ';'                                                     ),
                        fcfillStr(TO_STRING(tValue),GlobalKonstant.usiFeldLeng) ),
                        ';'                                                     ),
                        fcfillStr(TO_STRING(tMin),GlobalKonstant.usiFeldLeng)   ),
                        ';'                                                     ),
                        fcfillStr(TO_STRING(tMax),GlobalKonstant.usiFeldLeng)   );
END_GET
SET
proMax    := TO_TIME(fcGetMax  ( proStrPara));
proMin    := TO_TIME(fcGetMin  ( proStrPara));
proValue  := TO_TIME(fcGetValue( proStrPara));
END_SET
END_PROPERTY

PROPERTY proShowValue : STRING[40]
GET
proShowValue := TO_STRING(tValue);
END_GET
END_PROPERTY

METHOD metNewValueNoSave : BOOL
VAR_INPUT
    newValueNoSave   :   TIME;
END_VAR
proValue := newValueNoSave;
scState.xUpdateOldValueNoSave := TRUE;
metNewValueNoSave := TRUE;
END_METHOD

METHOD metNewValue : BOOL
VAR_INPUT
    newValue   :   TIME;
END_VAR
proValue := newValue;
metNewValue := TRUE;
END_METHOD

{attribute 'hide'}
METHOD metInit : BOOL
IF _MinInit <> _MaxInit THEN
    proMin    := _MinInit;
    proMax    := _MaxInit;
ELSE
    proMin    := T#0D0H0M0S0MS;
    proMax    := T#49D17H2M47S295MS;
END_IF;
    proValue  := _WertInit;
END_METHOD

METHOD metNewMinMax : BOOL
VAR_INPUT
    newMin      :   TIME;
    newMax      :   TIME;
END_VAR
IF newMin <> newMax THEN
    proMin      := newMin;
    proMax      := newMax;
    proValue    := tValue;    
END_IF;
metNewMinMax := TRUE;
END_METHOD

{attribute 'monitoring':='call'}
PROPERTY proMin : TIME
GET
proMin := tMin;
END_GET
SET
tMin := LIMIT(T#0D0H0M0S0MS,proMin,T#49D17H2M47S295MS);
END_SET
END_PROPERTY

METHOD metNewMinMaxNoSave : BOOL
VAR_INPUT
    newMinNoSave      :   TIME;
    newMaxNoSave      :   TIME;
END_VAR
IF newMinNoSave <> newMaxNoSave THEN
    proMin      := newMinNoSave;
    proMax      := newMaxNoSave;
    proValue    := tValue;    
    scState.xUpdateOldValueNoSave := TRUE;
END_IF;
metNewMinMaxNoSave := TRUE;
END_METHOD

{attribute 'monitoring':='call'}
PROPERTY proMax : TIME
SET
tMax := LIMIT(T#0D0H0M0S0MS,proMax,T#49D17H2M47S295MS);
END_SET
GET
proMax := tMax;
END_GET
END_PROPERTY

{attribute 'hide'}
METHOD metCheckState : BOOL
(* Search Change & Save Old Values *)
IF tValue <> tValueOld OR tMin <> tMinOld OR tMax <> tMaxOld OR scState.xUpdateOldValueNoSave THEN
    (* Prüfen ob die Werte bei änderung gespeichert werden sollen *)
    IF scState.xUpdateOldValueNoSave THEN
        scState.xUpdateOldValueNoSave := FALSE;
    ELSE
        proSaveOnChange 	:= TRUE;
	END_IF
	(*State Changed*) 
	scState.xStateChanged 	:= TRUE;   
    proValue  				:= tValue;
    tValueOld 				:= proValue;
    proMin    				:= tMin;
    proMax    				:= tMax;        
    tMinOld   				:= proMin;
    tMaxOld   				:= proMax;
ELSE
	(*State Changed*) 
	scState.xStateChanged 	:= FALSE;    
END_IF;
END_METHOD

END_FUNCTION_BLOCK

// 30 Program Organization Units/Functions/fcRealToString
FUNCTION fcRealToString : STRING
VAR_INPUT
    rIn             :   REAL;
    usiNachkomma    :   USINT;
END_VAR
VAR
    iFor            :   INT;
END_VAR

fcRealToString := TO_STRING(rIn);
IF usiNachkomma > 0 THEN
    IF FIND(fcRealToString,'E') = 0 THEN
        fcRealToString := DELETE(fcRealToString,LEN(fcRealToString)-(FIND(fcRealToString,'.')+usiNachkomma),(FIND(fcRealToString,'.')+usiNachkomma)+ 1);
        FOR iFor := 0 TO usiNachkomma - 1 DO
            IF RIGHT(fcRealToString,1) = '0' AND RIGHT(fcRealToString,2) <> '.0' THEN
                fcRealToString := DELETE(fcRealToString,1,LEN(fcRealToString));
            ELSE
                EXIT;
            END_IF;    
        END_FOR
    ELSE
        fcRealToString := TO_STRING(rIn); 
    END_IF;
END_IF;

END_FUNCTION

// 30 Program Organization Units/08 Bit/fbUSINT
FUNCTION_BLOCK fbUSINT EXTENDS fbDataType IMPLEMENTS ITF_USINT
VAR_INPUT CONSTANT
    _WertInit      :   USINT;
    _MinInit       :   UsINT;
    _MaxInit       :   UsINT;       
END_VAR
VAR
    usiValue          :   USINT;   
    usiMin            :   USINT;
    usiMax            :   USINT; 
    {attribute 'hide'}
    usiValueOld       :   USINT; 
    {attribute 'hide'}
    usiMinOld         :   USINT;
    {attribute 'hide'}
    usiMaxOld         :   USINT;
END_VAR

(* Call Supper Objekt *)
IF itfConfigFb <> 0 THEN
    SUPER^();
END_IF;

{attribute 'monitoring':='call'}
PROPERTY proMax : UsINT
GET
proMax := usiMax;
END_GET
SET
usiMax := LIMIT(0,proMax,255);
END_SET
END_PROPERTY

METHOD metNewValueNoSave : BOOL
VAR_INPUT
    newValueNoSave   :   USINT;
END_VAR
proValue := newValueNoSave;
scState.xUpdateOldValueNoSave := TRUE;
metNewValueNoSave := TRUE;
END_METHOD

{attribute 'hide'}
{attribute 'monitoring':='call'}
PROPERTY proStrPara : STRING(129)
// {attribute 'hide'}
GET
proStrPara :=   CONCAT(                    
                CONCAT( 
                CONCAT(
                CONCAT(                 
                CONCAT(                     
                CONCAT( fcfillStr(CONCAT('P',TO_STRING(SUPER^._usiParaNr)),6)       ,
                        ';'                                                         ),
                        fcfillStr(TO_STRING(usiValue),GlobalKonstant.usiFeldLeng)   ),
                        ';'                                                         ),
                        fcfillStr(TO_STRING(usiMin),GlobalKonstant.usiFeldLeng)     ),
                        ';'                                                         ),
                        fcfillStr(TO_STRING(usiMax),GlobalKonstant.usiFeldLeng)     );
END_GET
SET
proMax    := TO_USINT(fcGetMax  ( proStrPara));
proMin    := TO_USINT(fcGetMin  ( proStrPara));
proValue  := TO_USINT(fcGetValue( proStrPara));
END_SET
END_PROPERTY

{attribute 'hide'}
METHOD metInit : BOOL
IF _MinInit <> _MaxInit THEN
    proMin    := _MinInit;
    proMax    := _MaxInit;
ELSE
    proMin    := 0;
    proMax    := 255;
END_IF;
    proValue  := _WertInit;
END_METHOD

PROPERTY proShowValue : STRING[40]
GET
proShowValue := TO_STRING(usiValue);
END_GET
END_PROPERTY

METHOD metNewMinMaxNoSave : BOOL
VAR_INPUT
    newMinNoSave      :   USINT;
    newMaxNoSave      :   USINT;
END_VAR
IF newMinNoSave <> newMaxNoSave THEN
    proMin      := newMinNoSave;
    proMax      := newMaxNoSave;
    proValue    := usiValue;    
    scState.xUpdateOldValueNoSave := TRUE;
END_IF;
metNewMinMaxNoSave := TRUE;
END_METHOD

{attribute 'monitoring':='call'}
PROPERTY proValue : UsINT
SET
usiValue := LIMIT(proMin,proValue,proMax);
END_SET
GET
proValue := usiValue;
END_GET
END_PROPERTY

{attribute 'monitoring':='call'}
PROPERTY proMin : UsINT
SET
usiMin := LIMIT(0,proMin,255);
END_SET
GET
proMin := usiMin;
END_GET
END_PROPERTY

METHOD metNewMinMax : BOOL
VAR_INPUT
    newMin      :   USINT;
    newMax      :   USINT;
END_VAR
IF newMin <> newMax THEN
    proMin      := newMin;
    proMax      := newMax;
    proValue    := usiValue;    
END_IF;
metNewMinMax := TRUE;
END_METHOD

METHOD metNewValue : BOOL
VAR_INPUT
    newValue   :   USINT;
END_VAR
proValue := newValue;
metNewValue := TRUE;
END_METHOD

{attribute 'hide'}
METHOD metCheckState : BOOL
(* Search Change & Save Old Values *)
IF usiValue <> usiValueOld OR usiMin <> usiMinOld OR usiMax <> usiMaxOld OR scState.xUpdateOldValueNoSave THEN
    (* Prüfen ob die Werte bei änderung gespeichert werden sollen *)
    IF scState.xUpdateOldValueNoSave THEN
        scState.xUpdateOldValueNoSave := FALSE;
    ELSE
        proSaveOnChange 	:= TRUE;
	END_IF
	(*State Changed*) 
	scState.xStateChanged 	:= TRUE;   
    proValue    			:= usiValue;
    usiValueOld 			:= proValue;
    proMin      			:= usiMin;
    proMax      			:= usiMax;        
    usiMinOld   			:= proMin;
    usiMaxOld   			:= proMax;
ELSE
	(*State Changed*) 
	scState.xStateChanged 	:= FALSE;    
END_IF;
END_METHOD

END_FUNCTION_BLOCK

// 21 Interface/08 Bit/ITF_USINT
INTERFACE ITF_USINT EXTENDS ITF_DATATYPE

{attribute 'monitoring':='call'}
PROPERTY proMin : UsINT
SET
END_SET
GET
END_GET
END_PROPERTY

{attribute 'monitoring':='call'}
PROPERTY proValue : UsINT
SET
END_SET
GET
END_GET
END_PROPERTY

{attribute 'monitoring':='call'}
PROPERTY proMax : UsINT
SET
END_SET
GET
END_GET
END_PROPERTY

END_INTERFACE

// 30 Program Organization Units/Functions/fcGetEnumerationId
FUNCTION fcGetEnumerationId : DINT
VAR_INPUT
    visfbENUIn 	:	ITF_DATATYPE;	
END_VAR
VAR
	visfbBOOL	:	ITF_BOOL;
    visfbINT   	:   ITF_INT;	
    visfbDINT  	:   ITF_DINT;
END_VAR

IF __QUERYINTERFACE(visfbENUIn,visfbBOOL) THEN
	fcGetEnumerationId := TO_DINT(visfbBOOL.proValue);
ELSIF __QUERYINTERFACE(visfbENUIn,visfbINT) THEN
    fcGetEnumerationId := TO_DINT(visfbINT.proValue);    
ELSIF __QUERYINTERFACE(visfbENUIn,visfbDINT) THEN
    fcGetEnumerationId := visfbDINT.proValue;     
ELSE
    fcGetEnumerationId := 0;
END_IF;

END_FUNCTION

// 21 Interface/32 Bit/ITF_DINT
INTERFACE ITF_DINT EXTENDS ITF_DATATYPE

{attribute 'monitoring':='call'}
PROPERTY proMax : dINT
GET
END_GET
SET
END_SET
END_PROPERTY

{attribute 'monitoring':='call'}
PROPERTY proMin : dINT
GET
END_GET
SET
END_SET
END_PROPERTY

{attribute 'monitoring':='call'}
PROPERTY proValue : dINT
GET
END_GET
SET
END_SET
END_PROPERTY

END_INTERFACE

// 30 Program Organization Units/Basis/fbBackUpConfig
FUNCTION_BLOCK fbBackUpConfig
VAR_INPUT
END_VAR
VAR_OUTPUT
END_VAR
VAR
    xSave               :   BOOL;   
    xLoad               :   BOOL;
    xDelete             :   BOOL;
	{attribute 'monitoring_encoding' := 'UTF-8'}
    stFilePathAktual    :   STRING[255];    
	{attribute 'monitoring_encoding' := 'UTF-8'}
    stFilePathBackUp    :   STRING[255];    
	{attribute 'monitoring_encoding' := 'UTF-8'}
    stFilePathBackUp1   :   STRING[30] := 'Actual';  
    xCopy               :   BOOL;
    pResutl             :   RTS_IEC_RESULT;
    ayBackUpDate        :   ARRAY[0..6] OF STRING[19] := ['Actual Config', 6('')];
    stHS                    :   STRING[1]   :=  '#';            //  Hashtag
    stPP                    :   STRING[1]   :=  ':';            //  Doppelpunkt
    stSL                    :   STRING[1]   :=  '_';            //  Subline
    stMS                    :   STRING[1]   :=  '-';            //  Minus
    stSP                    :   STRING[1]   :=  ' ';            //  Space
    uiFor                   :   UINT;                           //  Forschleifen Variable für Sonderzeichen entfernen
	xRecursive: BOOL;
	xOverwrite: BOOL;
	pulCopied: DWORD;
    stDate              :   STRING[19];                     //  String mit dem aktuellen Datum ohne # und -
END_VAR

actCreateDateTime();
actCreateFilePath();
GVL_Config.xSave := FALSE;
IF xSave THEN
    GVL_Config.xSave := TRUE;
    GVL_Config.stBackUp := CONCAT(CONCAT('BackUp/',stDate),'/');
    ayBackUpDate[1]:= stDate;
END_IF;
xSave := FALSE;
IF xLoad THEN
    stFilePathBackUp := CONCAT(stFilePathBackUp,ayBackUpDate[1]);
END_IF;
IF xDelete THEN
    ;
END_IF

ACTION actCreateDateTime:
// String Cleaning
stDate      := '';
// Datum und Zeit auslesen
stDate := TO_STRING(FuGetLocalDateAndTime());
// Datum und Zeit für BackUp erstellen Format DT_2020_12_31_23h59
FOR uiFor := 0 TO SIZEOF(stDate)-1 DO
    // # und - durch _ ersetzen
    IF stDate[uiFor] = stHS[0] OR stDate[uiFor] = stMS[0] OR stDate[uiFor] = stSP[0] THEN
        stDate[uiFor] := stSL[0];
    END_IF; 
    // Doppelpunkt durch h ersetzen und Sekunden löschen
    IF stDate[uiFor] = stPP[0] THEN
        stDate := REPLACE(stDate,'h',1,TO_INT(uiFor+1));  
        stDate := DELETE(stDate,TO_INT(SIZEOF(stDate)-uiFor+2),TO_INT(uiFor+4)); 
        EXIT;
    END_IF;    
END_FOR;
END_ACTION

ACTION actCreateFilePath:
{IF NOT defined (IsSimulationMode)}
    // FILE Path auf SPS
	stFilePathAktual      :=  CONCAT(                            
                                        './',
                                        'ConfigFiles/Actual/');   
	
	stFilePathBackUp      :=  CONCAT(                            
                                        './',
                                        'ConfigFiles/BackUp/');       
    {ELSE}
    // FILE Path auf Laptop
    stFilePathAktual      :=  'C:\PFC_Simulation\ConfigFiles\Actual\';  

    stFilePathBackUp      :=  'C:\PFC_Simulation\ConfigFiles\BackUp\';                                                         
{END_IF}
END_ACTION

END_FUNCTION_BLOCK

// 30 Program Organization Units/FuGetLocalDateAndTime
FUNCTION FuGetLocalDateAndTime : DT
VAR_INPUT
END_VAR
VAR
	RTS_RESULT	:	SysTypes.RTS_IEC_RESULT;
	dwTemp		:	DWORD;
END_VAR

RTS_RESULT := SysTimeRtc.SysTimeRtcConvertUtcToLocal(SysTimeRtc.SysTimeRtcGet(RTS_RESULT),dwTemp);
FuGetLocalDateAndTime := TO_DT(dwTemp);

END_FUNCTION

// 30 Program Organization Units/32 Bit/fbDINT
FUNCTION_BLOCK fbDINT EXTENDS fbDataType IMPLEMENTS ITF_DINT
VAR_INPUT CONSTANT 
    _WertInit      :   DINT;
    _MinInit       :   DINT;
    _MaxInit       :   DINT;      
END_VAR
VAR
    diValue          :   DINT;
    diMin            :   DINT;
    diMax            :   DINT;
    {attribute 'hide'}
    diValueOld       :   DINT;
    {attribute 'hide'}
    diMinOld         :   DINT;
    {attribute 'hide'}
    diMaxOld         :   DINT;
END_VAR

(* Call Supper Objekt *)
IF itfConfigFb <> 0 THEN
    SUPER^();
END_IF;

{attribute 'hide'}
{attribute 'monitoring':='call'}
PROPERTY proStrPara : STRING(129)
// {attribute 'hide'}
SET
proMax    := TO_DINT(fcGetMax  ( proStrPara));
proMin    := TO_DINT(fcGetMin  ( proStrPara));
proValue  := TO_DINT(fcGetValue( proStrPara));
END_SET
GET
proStrPara :=   CONCAT(                    
                CONCAT( 
                CONCAT(
                CONCAT(                 
                CONCAT(                     
                CONCAT( fcfillStr(CONCAT('P',TO_STRING(SUPER^._usiParaNr)),6)       ,
                        ';'                                                         ),
                        fcfillStr(TO_STRING(diValue),GlobalKonstant.usiFeldLeng)    ),
                        ';'                                                         ),
                        fcfillStr(TO_STRING(diMin),GlobalKonstant.usiFeldLeng)      ),
                        ';'                                                         ),
                        fcfillStr(TO_STRING(diMax),GlobalKonstant.usiFeldLeng)      );
END_GET
END_PROPERTY

{attribute 'hide'}
METHOD metInit : BOOL
IF _MinInit <> _MaxInit THEN
    proMin    := _MinInit;
    proMax    := _MaxInit;
ELSE
    proMin    := -2147483648;
    proMax    :=  2147483647;
END_IF;
    proValue  := _WertInit;
END_METHOD

METHOD metNewValue : BOOL
VAR_INPUT
    newValue   :   DINT;
END_VAR
proValue := newValue;
metNewValue := TRUE;
END_METHOD

{attribute 'monitoring':='call'}
PROPERTY proValue : dINT
SET
diValue := LIMIT(proMin,proValue,proMax);
END_SET
GET
proValue := diValue;
END_GET
END_PROPERTY

METHOD metNewMinMax : BOOL
VAR_INPUT
    newMin      :   DINT;
    newMax      :   DINT;
END_VAR
IF newMin <> newMax THEN
    proMin      := newMin;
    proMax      := newMax;
    proValue    := diValue;    
END_IF;
metNewMinMax := TRUE;
END_METHOD

{attribute 'monitoring':='call'}
PROPERTY proMin : dINT
SET
diMin := LIMIT(-2147483648,proMin,2147483647);
END_SET
GET
proMin := diMin;
END_GET
END_PROPERTY

METHOD metNewMinMaxNoSave : BOOL
VAR_INPUT
    newMinNoSave      :   DINT;
    newMaxNoSave      :   DINT;
END_VAR
IF newMinNoSave <> newMaxNoSave THEN
    proMin      := newMinNoSave;
    proMax      := newMaxNoSave;
    proValue    := diValue;    
    scState.xUpdateOldValueNoSave := TRUE;
END_IF;
metNewMinMaxNoSave := TRUE;
END_METHOD

{attribute 'monitoring':='call'}
PROPERTY proMax : dINT
SET
diMax := LIMIT(-2147483648,proMax,2147483647);
END_SET
GET
proMax := diMax;
END_GET
END_PROPERTY

PROPERTY proShowValue : STRING[40]
GET
proShowValue := TO_STRING(diValue);
END_GET
END_PROPERTY

METHOD metNewValueNoSave : BOOL
VAR_INPUT
    newValueNoSave   :   DINT;
END_VAR
proValue := newValueNoSave;
scState.xUpdateOldValueNoSave := TRUE;
metNewValueNoSave := TRUE;
END_METHOD

{attribute 'hide'}
METHOD metCheckState : BOOL
(* Search Change & Save Old Values *)
IF diValue <> diValueOld OR diMin <> diMinOld OR diMax <> diMaxOld OR scState.xUpdateOldValueNoSave THEN
    (* Prüfen ob die Werte bei änderung gespeichert werden sollen *)
    IF scState.xUpdateOldValueNoSave THEN
        scState.xUpdateOldValueNoSave := FALSE;
    ELSE
        proSaveOnChange 	:= TRUE;
	END_IF
	(*State Changed*) 
	scState.xStateChanged 	:= TRUE;   
    proValue   				:= diValue;
    diValueOld 				:= proValue;
    proMin     				:= diMin;
    proMax     				:= diMax;        
    diMinOld   				:= proMin;
    diMaxOld   				:= proMax;
ELSE
	(*State Changed*) 
	scState.xStateChanged 	:= FALSE;    
END_IF;
END_METHOD

END_FUNCTION_BLOCK

// 21 Interface/40 Byte String/ITF_STRING40
INTERFACE ITF_STRING40 EXTENDS ITF_DATATYPE

{attribute 'monitoring':='call'}
{attribute 'monitoring_encoding' := 'UTF-8'}
PROPERTY proValue : STRING[40]
SET
END_SET
GET
END_GET
END_PROPERTY

END_INTERFACE

// 30 Program Organization Units/32 Bit/fbTOD
FUNCTION_BLOCK fbTOD EXTENDS fbDataType IMPLEMENTS ITF_TOD
VAR_INPUT CONSTANT 
    _WertInit        :   TOD;
    _MinInit         :   TOD;
    _MaxInit       	 :   TOD;      
END_VAR
VAR
    todValue         :   TOD;
    todMin           :   TOD;
    todMax           :   TOD;
    {attribute 'hide'}
    todValueOld      :   TOD;
    {attribute 'hide'}
    todMinOld        :   TOD;
    {attribute 'hide'}
    todMaxOld        :   TOD;
END_VAR

(* Call Supper Objekt *)
IF itfConfigFb <> 0 THEN
    SUPER^();
END_IF;

{attribute 'hide'}
{attribute 'monitoring':='call'}
PROPERTY proStrPara : STRING(129)
// {attribute 'hide'}
SET
proMax    := TO_TOD(fcGetMax  ( proStrPara));
proMin    := TO_TOD(fcGetMin  ( proStrPara));
proValue  := TO_TOD(fcGetValue( proStrPara));
END_SET
GET
proStrPara :=   CONCAT(                    
                CONCAT( 
                CONCAT(
                CONCAT(                 
                CONCAT(                     
                CONCAT( fcfillStr(CONCAT('P',TO_STRING(SUPER^._usiParaNr)),6)       ,
                        ';'                                                         ),
                        fcfillStr(TO_STRING(todValue),GlobalKonstant.usiFeldLeng)    ),
                        ';'                                                         ),
                        fcfillStr(TO_STRING(todMin),GlobalKonstant.usiFeldLeng)      ),
                        ';'                                                         ),
                        fcfillStr(TO_STRING(todMax),GlobalKonstant.usiFeldLeng)      );
END_GET
END_PROPERTY

{attribute 'hide'}
METHOD metInit : BOOL
IF _MinInit <> _MaxInit THEN
    proMin    := _MinInit;
    proMax    := _MaxInit;
ELSE
    proMin    := TOD#00:00:00;
    proMax    := TOD#23:59:59;
END_IF;
    proValue  := _WertInit;
END_METHOD

METHOD metNewMinMax : BOOL
VAR_INPUT
    newMin      :   TOD;
    newMax      :   TOD;
END_VAR
IF newMin <> newMax THEN
    proMin      := newMin;
    proMax      := newMax;
    proValue    := todValue;    
END_IF;
metNewMinMax := TRUE;
END_METHOD

{attribute 'monitoring':='call'}
PROPERTY proMin : TOD
GET
proMin := todMin;
END_GET
SET
todMin := LIMIT(TOD#00:00:00,proMin,TOD#23:59:59);
END_SET
END_PROPERTY

{attribute 'monitoring':='call'}
PROPERTY proValue : TOD
GET
proValue := todValue;
END_GET
SET
todValue := LIMIT(proMin,proValue,proMax);
END_SET
END_PROPERTY

METHOD metNewValueNoSave : BOOL
VAR_INPUT
    newValueNoSave   :   TOD;
END_VAR
proValue := newValueNoSave;
scState.xUpdateOldValueNoSave := TRUE;
metNewValueNoSave := TRUE;
END_METHOD

METHOD metNewMinMaxNoSave : BOOL
VAR_INPUT
    newMinNoSave      :   TOD;
    newMaxNoSave      :   TOD;
END_VAR
IF newMinNoSave <> newMaxNoSave THEN
    proMin      := newMinNoSave;
    proMax      := newMaxNoSave;
    proValue    := todValue;    
    scState.xUpdateOldValueNoSave := TRUE;
END_IF;
metNewMinMaxNoSave := TRUE;
END_METHOD

METHOD metNewValue : BOOL
VAR_INPUT
    newValue   :   TOD;
END_VAR
proValue := newValue;
metNewValue := TRUE;
END_METHOD

PROPERTY proShowValue : STRING[40]
GET
proShowValue := TO_STRING(todValue);
END_GET
END_PROPERTY

{attribute 'monitoring':='call'}
PROPERTY proMax : TOD
SET
todMax := LIMIT(TOD#00:00:00,proMax,TOD#23:59:59);
END_SET
GET
proMax := todMax;
END_GET
END_PROPERTY

{attribute 'hide'}
METHOD metCheckState : BOOL
(* Search Change & Save Old Values *)
IF todValue <> todValueOld OR todMin <> todMinOld OR todMax <> todMaxOld OR scState.xUpdateOldValueNoSave THEN
    (* Prüfen ob die Werte bei änderung gespeichert werden sollen *)
    IF scState.xUpdateOldValueNoSave THEN
        scState.xUpdateOldValueNoSave := FALSE;
    ELSE
        proSaveOnChange 	:= TRUE;
	END_IF
	(*State Changed*) 
	scState.xStateChanged 	:= TRUE;   
    proValue   				:= todValue;
    todValueOld 			:= proValue;
    proMin     				:= todMin;
    proMax     				:= todMax;        
    todMinOld   			:= proMin;
    todMaxOld   			:= proMax;
ELSE
	(*State Changed*) 
	scState.xStateChanged 	:= FALSE;    
END_IF;
END_METHOD

END_FUNCTION_BLOCK

// 30 Program Organization Units/32 Bit/fbDATE_AND_TIME
FUNCTION_BLOCK fbDATE_AND_TIME EXTENDS fbDataType IMPLEMENTS ITF_DATE_AND_TIME
VAR_INPUT CONSTANT
    _WertInit       :   DT;
    _MinInit        :   DT;
    _MaxInit        :   DT;       
END_VAR
VAR
    dtValue         :   DT;   
    dtMin           :   DT;
    dtMax           :   DT; 
    {attribute 'hide'}
    dtValueOld      :   DT;
    {attribute 'hide'}
    dtMinOld        :   DT;
    {attribute 'hide'}
    dtMaxOld        :   DT;
END_VAR

(* Call Supper Objekt *)
IF itfConfigFb <> 0 THEN
    SUPER^();
END_IF;

METHOD metNewMinMax : BOOL
VAR_INPUT
    newMin      :   DT;
    newMax      :   DT;
END_VAR
IF newMin <> newMax THEN
    proMin      := newMin;
    proMax      := newMax;
    proValue    := dtValue;    
END_IF;
metNewMinMax := TRUE;
END_METHOD

{attribute 'monitoring':='call'}
PROPERTY proMax : DT
SET
dtMax := LIMIT(DT#1970-01-01-00:00:00,proMax,DT#2106-02-07-06:28:15);
END_SET
GET
proMax := dtMax;
END_GET
END_PROPERTY

{attribute 'hide'}
{attribute 'monitoring':='call'}
PROPERTY proStrPara : STRING[129]
SET
proMax    := TO_DT(fcGetMax  ( proStrPara));
proMin    := TO_DT(fcGetMin  ( proStrPara));
proValue  := TO_DT(fcGetValue( proStrPara));
END_SET
GET
proStrPara :=   CONCAT(                    
                CONCAT( 
                CONCAT(
                CONCAT(                 
                CONCAT(                  
                CONCAT( fcfillStr(CONCAT('P',TO_STRING(SUPER^._usiParaNr)),6)   ,
                        ';'                                                     ),
                        fcfillStr(TO_STRING(dtValue),GlobalKonstant.usiFeldLeng)),
                        ';'                                                     ),
                        fcfillStr(TO_STRING(dtMin),GlobalKonstant.usiFeldLeng)  ),
                        ';'                                                     ),
                        fcfillStr(TO_STRING(dtMax),GlobalKonstant.usiFeldLeng)  );
END_GET
END_PROPERTY

{attribute 'monitoring':='call'}
PROPERTY proValue : DT
SET
dtValue := LIMIT(proMin,proValue,proMax);
END_SET
GET
proValue := LIMIT(dtMin,dtValue,dtMax);
END_GET
END_PROPERTY

{attribute 'hide'}
METHOD metInit : BOOL
IF _MinInit <> _MaxInit THEN
    proMin    := _MinInit;
    proMax    := _MaxInit;
ELSE
    proMin    := DT#1970-01-01-00:00:00;
    proMax    := DT#2106-02-07-06:28:15;
END_IF;
    proValue  := _WertInit;
END_METHOD

PROPERTY proShowValue : STRING[40]
GET
proShowValue := TO_STRING(dtValue);
END_GET
END_PROPERTY

METHOD metNewMinMaxNoSave : BOOL
VAR_INPUT
    newMinNoSave      :   DT;
    newMaxNoSave      :   DT;
END_VAR
IF newMinNoSave <> newMaxNoSave THEN
    proMin      := newMinNoSave;
    proMax      := newMaxNoSave;
    proValue    := dtValue;    
    scState.xUpdateOldValueNoSave := TRUE;
END_IF;
metNewMinMaxNoSave := TRUE;
END_METHOD

{attribute 'monitoring':='call'}
PROPERTY proMin : DT
GET
proMin := dtMin;
END_GET
SET
dtMin := LIMIT(DT#1970-01-01-00:00:00,proMin,DT#2106-02-07-06:28:15);
END_SET
END_PROPERTY

METHOD metNewValue : BOOL
VAR_INPUT
    newValue   :   DT;
END_VAR
proValue := newValue;
metNewValue := TRUE;
END_METHOD

METHOD metNewValueNoSave : BOOL
VAR_INPUT
    newValueNoSave   :   DT;
END_VAR
proValue := newValueNoSave;
scState.xUpdateOldValueNoSave := TRUE;
metNewValueNoSave := TRUE;
END_METHOD

{attribute 'hide'}
METHOD metCheckState : BOOL
(* Search Change & Save Old Values *)
IF dtValue <> dtValueOld OR dtMin <> dtMinOld OR dtMax <> dtMaxOld OR scState.xUpdateOldValueNoSave THEN
    (* Prüfen ob die Werte bei änderung gespeichert werden sollen *)
    IF scState.xUpdateOldValueNoSave THEN
        scState.xUpdateOldValueNoSave := FALSE;
    ELSE
        proSaveOnChange 	:= TRUE;
	END_IF
	(*State Changed*) 
	scState.xStateChanged 	:= TRUE;   
    proValue    			:= dtValue;
    dtValueOld  			:= proValue;
    proMin      			:= dtMin;
    proMax      			:= dtMax;        
    dtMinOld    			:= proMin;
    dtMaxOld    			:= proMax;
ELSE
	(*State Changed*) 
	scState.xStateChanged 	:= FALSE;    
END_IF;
END_METHOD

END_FUNCTION_BLOCK

// 30 Program Organization Units/64 Bit/fbLTIME
FUNCTION_BLOCK fbLTIME EXTENDS fbDataType IMPLEMENTS ITF_LTIME
VAR_INPUT CONSTANT
    _WertInit      :   LTIME;
    _MinInit       :   LTIME;
    _MaxInit       :   LTIME;       
END_VAR
VAR
    tValue          :   LTIME;   
    tMin            :   LTIME;
    tMax            :   LTIME; 
    {attribute 'hide'}
    tValueOld       :   LTIME;
    {attribute 'hide'}
    tMinOld         :   LTIME;
    {attribute 'hide'}
    tMaxOld         :   LTIME;
END_VAR

(* Call Supper Objekt *)
IF itfConfigFb <> 0 THEN
    SUPER^();
END_IF;

{attribute 'monitoring':='call'}
PROPERTY proValue : LTIME
GET
proValue := LIMIT(tMin,tValue,tMax);
END_GET
SET
tValue := LIMIT(proMin,proValue,proMax);
END_SET
END_PROPERTY

METHOD metNewValue : BOOL
VAR_INPUT
    newValue   :   LTIME;
END_VAR
proValue := newValue;
metNewValue := TRUE;
END_METHOD

{attribute 'hide'}
METHOD metInit : BOOL
IF _MinInit <> _MaxInit THEN
    proMin    := _MinInit;
    proMax    := _MaxInit;
ELSE
    proMin    := LTIME#0NS;
    proMax    := LTIME#213503D23H34M33S709MS551US615NS;
END_IF;
    proValue  := _WertInit;
END_METHOD

{attribute 'monitoring':='call'}
PROPERTY proMin : LTIME
SET
tMin := LIMIT(LTIME#0NS,proMin,LTIME#213503D23H34M33S709MS551US615NS);
END_SET
GET
proMin := tMin;
END_GET
END_PROPERTY

METHOD metNewValueNoSave : BOOL
VAR_INPUT
    newValueNoSave   :   LTIME;
END_VAR
proValue := newValueNoSave;
scState.xUpdateOldValueNoSave := TRUE;
metNewValueNoSave := TRUE;
END_METHOD

PROPERTY proShowValue : STRING[40]
GET
proShowValue := TO_STRING(tValue);
END_GET
END_PROPERTY

METHOD metNewMinMax : BOOL
VAR_INPUT
    newMin      :   LTIME;
    newMax      :   LTIME;
END_VAR
IF newMin <> newMax THEN
    proMin      := newMin;
    proMax      := newMax;
    proValue    := tValue;    
END_IF;
metNewMinMax := TRUE;
END_METHOD

{attribute 'hide'}
{attribute 'monitoring':='call'}
PROPERTY proStrPara : STRING[129]
GET
proStrPara :=   CONCAT(                    
                CONCAT( 
                CONCAT(
                CONCAT(                 
                CONCAT(                  
                CONCAT( fcfillStr(CONCAT('P',TO_STRING(SUPER^._usiParaNr)),6)    ,
                        ';'                                                     ),
                        fcfillStr(TO_STRING(tValue),GlobalKonstant.usiFeldLeng) ),
                        ';'                                                     ),
                        fcfillStr(TO_STRING(tMin),GlobalKonstant.usiFeldLeng)   ),
                        ';'                                                     ),
                        fcfillStr(TO_STRING(tMax),GlobalKonstant.usiFeldLeng)   );
END_GET
SET
proMax    := TO_LTIME(fcGetMax  ( proStrPara));
proMin    := TO_LTIME(fcGetMin  ( proStrPara));
proValue  := TO_LTIME(fcGetValue( proStrPara));
END_SET
END_PROPERTY

{attribute 'monitoring':='call'}
PROPERTY proMax : LTIME
SET
tMax := LIMIT(LTIME#0NS,proMax,LTIME#213503D23H34M33S709MS551US615NS);
END_SET
GET
proMax := tMax;
END_GET
END_PROPERTY

METHOD metNewMinMaxNoSave : BOOL
VAR_INPUT
    newMinNoSave      :   LTIME;
    newMaxNoSave      :   LTIME;
END_VAR
IF newMinNoSave <> newMaxNoSave THEN
    proMin      := newMinNoSave;
    proMax      := newMaxNoSave;
    proValue    := tValue;    
    scState.xUpdateOldValueNoSave := TRUE;
END_IF;
metNewMinMaxNoSave := TRUE;
END_METHOD

{attribute 'hide'}
METHOD metCheckState : BOOL
(* Search Change & Save Old Values *)
IF tValue <> tValueOld OR tMin <> tMinOld OR tMax <> tMaxOld OR scState.xUpdateOldValueNoSave THEN
    (* Prüfen ob die Werte bei änderung gespeichert werden sollen *)
    IF scState.xUpdateOldValueNoSave THEN
        scState.xUpdateOldValueNoSave := FALSE;
    ELSE
        proSaveOnChange 	:= TRUE;
	END_IF
	(*State Changed*) 
	scState.xStateChanged 	:= TRUE;   
    proValue  				:= tValue;
    tValueOld 				:= proValue;
    proMin    				:= tMin;
    proMax    				:= tMax;        
    tMinOld   				:= proMin;
    tMaxOld   				:= proMax;
ELSE
	(*State Changed*) 
	scState.xStateChanged 	:= FALSE;    
END_IF;
END_METHOD

END_FUNCTION_BLOCK

// 21 Interface/64 Bit/ITF_LTIME
INTERFACE ITF_LTIME EXTENDS ITF_DATATYPE

{attribute 'monitoring':='call'}
PROPERTY proValue : LTIME
GET
END_GET
SET
END_SET
END_PROPERTY

{attribute 'monitoring':='call'}
PROPERTY proMin : LTIME
SET
END_SET
GET
END_GET
END_PROPERTY

{attribute 'monitoring':='call'}
PROPERTY proMax : LTIME
SET
END_SET
GET
END_GET
END_PROPERTY

END_INTERFACE

// 30 Program Organization Units/Functions/fcFileDelete
FUNCTION fcFileDelete : RTS_IEC_HANDLE
VAR_INPUT
	{attribute 'monitoring_encoding' := 'UTF-8'}
    stFilePath  :   STRING[255];
END_VAR
VAR
    RTS_IEC_RESULT_DEL  :   RTS_IEC_RESULT;
	RTS_IEC_HANDLE_DEL	:	RTS_IEC_HANDLE;
END_VAR

RTS_IEC_RESULT_DEL := SysFile.SysFileDelete(stFilePath);

END_FUNCTION

// 30 Program Organization Units/Basis/fbConfigFile
{attribute 'enable_dynamic_creation'}
{attribute 'hide_all_locals'}
{attribute 'reflection'} 
FUNCTION_BLOCK fbConfigFile IMPLEMENTS ITF_CONFIGFILE
VAR_OUTPUT
    xError              :   BOOL;
    uiErrorNr           :   UINT;
END_VAR
VAR
    {attribute 'instance-path'} 
    {attribute 'noinit'}     
	{attribute 'monitoring_encoding' := 'UTF-8'}
    stCodeDir               :   STRING[255]; 
    iCaseInit               :   INT                 := 0;
    scState                 :   scStateConfigFile;
    hFile                   :   RTS_IEC_HANDLE;
    pResult                 :   RTS_IEC_RESULT;
    hFileCheck              :   RTS_IEC_HANDLE;
    pResultCheck            :   RTS_IEC_RESULT;    
	usiLastChild			:	USINT;
END_VAR

CASE iCaseInit OF
	0: // Get Last Child
		scState.xGetChild   := TRUE;
		metCodeDirCreate();
		iCaseInit := iCaseInit + 1;
	1: // Init
		scState.xGetChild	:= FALSE;
        scState.xInit       := TRUE;
		hFile := fcFileOpen(proFilePath,SysFile.ACCESS_MODE.AM_APPEND_PLUS,pResult);
		// Check File
		hFileCheck := fcFileOpen(proFilePathCheckFile,SysFile.ACCESS_MODE.AM_WRITE_PLUS,pResultCheck);
		iCaseInit   := iCaseInit + 1;
	2: // Init Done
		;	// Wait on Clean up Init Call
	3: // Check if Save or Load 
		IF (GVL_Config.xSave OR GVL_Config.xLoad) AND_THEN hFile = 0 THEN
            scState.xIsOpen := metOpenFile();  
		END_IF;
	ELSE
		iCaseInit   := 0;   
END_CASE;
// Meldung 
IF NOT scState.xEventLoad AND NOT scState.xEventSave AND scState.xEventDetekted THEN
	scState.xEventDetekted := FALSE; 
END_IF;
IF scState.xEventSave THEN
	scState.xEventDetekted := TRUE;
	scState.xEventSave 	   := FALSE;    
END_IF;    
IF scState.xEventLoad THEN
	scState.xEventDetekted := TRUE;
	scState.xEventLoad     := FALSE;    
END_IF; 
IF xError AND_THEN NOT GVL_Config.xError THEN
    GVL_Config.xError 	:= TRUE;
    GVL_Config.stPath	:= stCodeDir;
END_IF;

METHOD FINAL metLoad : BOOL
VAR_INPUT  
    itfDataTypeObj  :   ITF_DATATYPE;
END_VAR
VAR
    uiSafetyCount   :   UINT;
END_VAR
IF proLoad THEN
    REPEAT
        pResult       := 0;
        IF NOT scState.xIsOpen THEN
            scState.xIsOpen := metOpenFile();    
		END_IF
        IF scState.xIsOpen THEN
            metLoad       := metLoadFile(itfDataTypeObj);  
        END_IF;    
            uiSafetyCount := uiSafetyCount + 1;
    UNTIL
        metLoad = TRUE OR uiSafetyCount = 16#FFFF
    END_REPEAT;     
    IF NOT metLoad THEN
        THIS^.proError      := TRUE;
        THIS^.proErrorNr    := itfDataTypeObj.proParaNr;
    END_IF; 
END_IF;
END_METHOD

METHOD metOpenFile : BOOL
VAR_INPUT
END_VAR
hFile   := fcFileOpen(proFilePath,SysFile.ACCESS_MODE.AM_APPEND_PLUS,pResult);
presult := fcFileClose(hFile,stCodeDir,'FbConfigFile metOpenFile Z2');
hFile   := fcFileOpen(proFilePath,SysFile.ACCESS_MODE.AM_READ_PLUS,pResult);
IF pResult = 0 AND hFile <> 0 THEN
    metOpenFile := TRUE;
ELSE
    metOpenFile := FALSE;
END_IF
END_METHOD

PROPERTY proErrorNr : UINT
SET
uiErrorNr := proErrorNr;
END_SET
GET
proErrorNr := uiErrorNr;
END_GET
END_PROPERTY

METHOD PRIVATE FINAL metCodeDirCreate : BOOL
VAR
    uiFor                   :   UINT;
END_VAR
// Instanzpfad des Funktionsbausteinens in Ordnerstrucktur wandeln
FOR uiFor := 0 TO SIZEOF(stCodeDir)-1 DO
    // Punkt . durch Slash / ersetzen
    IF stCodeDir[uiFor] = 46 THEN
        stCodeDir[uiFor] := 47;
    END_IF;            
END_FOR;
END_METHOD

//FB_Exit muss explizit implementiert werden. Wenn es eine Implementierung gibt, dann wird 
//die Methode aufgerufen, bevor die Steuerung den Code der Funktionsbaustein-Instanz entfernt
//(impliziter Aufruf. Der Rückgabewert wird nicht ausgewertet.
METHOD FINAL FB_Exit: BOOL
VAR_INPUT    
    bInCopyCode: BOOL;  // TRUE: Die Exit-Methode wird aufgerufen, um die Instanz zu verlassen, die hinterher kopiert wird Online-Change).  
END_VAR
IF hFile <> 0 THEN
	pResult := SysFile.SysFileClose(hFile);
	hFile   := 0;
END_IF;
IF hFileCheck <> 0 THEN 
	SysFile.SysFileClose(hFileCheck);
	fcFileDelete(proFilePathCheckFile);
	hFileCheck  := 0;
END_IF;
END_METHOD

METHOD FINAL metLoadFile : BOOL
VAR_INPUT  
    itfDataTypeObj  :   ITF_DATATYPE;
END_VAR
VAR
    udiPos  : UDINT;
    stRead  : STRING[170];
    xValid  : BOOL;
END_VAR
IF hFile <> 0 AND itfDataTypeObj.proParaNr > 0 THEN
    udiPos := LIMIT(1,itfDataTypeObj.proParaNr,255);
   IF udiPos = 1 THEN
        udiPos :=  udiPos -1;   
    ELSE 
        udiPos := (udiPos * GlobalKonstant.diLineSize) - GlobalKonstant.diLineSize;
	END_IF;
    pResult := SysFile.SysFileSetPos(hFile,udiPos);
END_IF;
IF pResult = 0 AND hFile <> 0 THEN
    SysFile.SysFileRead(hFile,ADR(stRead),GlobalKonstant.diStringSize,ADR(pResult));
    stRead[170] := 0;
    IF itfDataTypeObj.proParaNr = TO_UINT(MID(stRead,5,2)) THEN
        itfDataTypeObj.proStrPara := stRead;
        xValid := TRUE;
	END_IF;
END_IF;
metLoadFile := NOT TO_BOOL(pResult) AND xValid;
scState.xEventLoad := TRUE;
END_METHOD

PROPERTY proEventDetekted : BOOL
GET
proEventDetekted := scState.xEventDetekted;
END_GET
END_PROPERTY

METHOD FINAL metCheckNr : BOOL
VAR_INPUT
    itfDataTypeObj  :   ITF_DATATYPE;
    xCheck          :   BOOL;
    xCheckDone      :   BOOL;
END_VAR
VAR
    udiPos  : UDINT;
    stReSa  : STRING[1];
    xValid  : BOOL;
    pulPos  : DWORD;
END_VAR
IF xCheck THEN
    IF pResultCheck = 0 AND itfDataTypeObj.proParaNr > 0 THEN
        udiPos := LIMIT(1,itfDataTypeObj.proParaNr,255)-1;
        pResultCheck := SysFile.SysFileSetPos(hFileCheck,udiPos);
    END_IF;
    IF pResultCheck = 0 THEN
        SysFile.SysFileRead(hFileCheck,ADR(stReSa),1,ADR(pResultCheck));
        IF TO_INT(stReSa) = 1 THEN
            xValid 		:= FALSE; 
			proError 	:= TRUE;
			proErrorNr 	:= itfDataTypeObj.proParaNr;
        ELSE
            xValid := TRUE; 
		END_IF
	ELSE
		proError := TRUE;
    END_IF;
    metCheckNr := NOT TO_BOOL(pResultCheck) AND xValid;
ELSIF xCheckDone THEN
    IF pResultCheck = 0 AND itfDataTypeObj.proParaNr > 0 THEN
            udiPos := LIMIT(1,itfDataTypeObj.proParaNr,255)-1;
            stReSa := TO_STRING(1);
            pResultCheck := SysFile.SysFileGetPos(hFile,ADR(pulPos));
            pResultCheck := SysFile.SysFileSetPos(hFile,udiPos);
            pResultCheck := SysFile.SysFileGetPos(hFile,ADR(pulPos));
    END_IF;
    IF pResultCheck = 0 THEN
        SysFile.SysFileWrite(hFileCheck,ADR(stReSa),TO_UINT(LEN(stReSa)),ADR(pResultCheck));
	ELSE
		proError := TRUE;	
    END_IF;    
END_IF;
END_METHOD

PROPERTY proFilePathCheckFile : STRING[255];
GET
// FILE Path auf SPS
 proFilePathCheckFile:= CONCAT(  
						CONCAT(  
						CONCAT(                                  
								'./',  
								'ConfigFiles/Actual/'),  
								stCodeDir),  
								'_Check.txt');
END_GET
END_PROPERTY

METHOD metChild
VAR_INPUT
	itfDataTypeObj  :   ITF_DATATYPE;
END_VAR
IF scState.xGetChild THEN
	IF __QUERYINTERFACE(itfDataTypeObj,itfDataTypeObj) THEN
		IF NOT itfDataTypeObj.proChildAddDone THEN
			usiLastChild := itfDataTypeObj.proparaNr;
			itfDataTypeObj.proChildAddDone := TRUE;
		END_IF;
	END_IF;
END_IF;
END_METHOD

{attribute 'monitoring':='call'}
PROPERTY proLoad : BOOL
GET
proLoad := GVL_Config.xLoad;
END_GET
END_PROPERTY

METHOD FINAL metSaveFile : BOOL
VAR_INPUT  
    itfDataTypeObj  :   ITF_DATATYPE;
END_VAR
VAR
    udiPos  : UDINT;
    stSave  : STRING[172];
	pulPos  : DWORD;
    dwWrite : DWORD;
END_VAR
IF hFile <> 0 AND pResult = 0 AND itfDataTypeObj.proParaNr > 0 THEN
    udiPos := LIMIT(1,itfDataTypeObj.proParaNr,255);
   IF udiPos = 1 THEN
        udiPos :=  udiPos -1;  
        stSave := CONCAT(itfDataTypeObj.proStrPara,'$R'); 
    ELSE
        udiPos := (udiPos * GlobalKonstant.diLineSize) - GlobalKonstant.diLineSize - 1;
        stSave := CONCAT('$N',CONCAT(itfDataTypeObj.proStrPara,'$R')); 
	END_IF;
        pResult := SysFile.SysFileGetPos(hFile,ADR(pulPos));
        pResult := SysFile.SysFileSetPos(hFile,udiPos);
        pResult := SysFile.SysFileGetPos(hFile,ADR(pulPos));
    IF hFile <> 0 AND pResult = 0 THEN
        dwWrite := TO_DWORD(SysFile.SysFileWrite(hFile,ADR(stSave),TO_UDINT(LEN(stSave)),ADR(pResult)));
    END_IF;
END_IF;
IF pResult <> 0 THEN
    pResult := pResult;
ELSE
    metSaveFile := NOT TO_BOOL(pResult) AND dwWrite = TO_UDINT(LEN(stSave));
END_IF
scState.xEventSave := TRUE;
END_METHOD

